ABB RAPID module: Robotpaint.mod

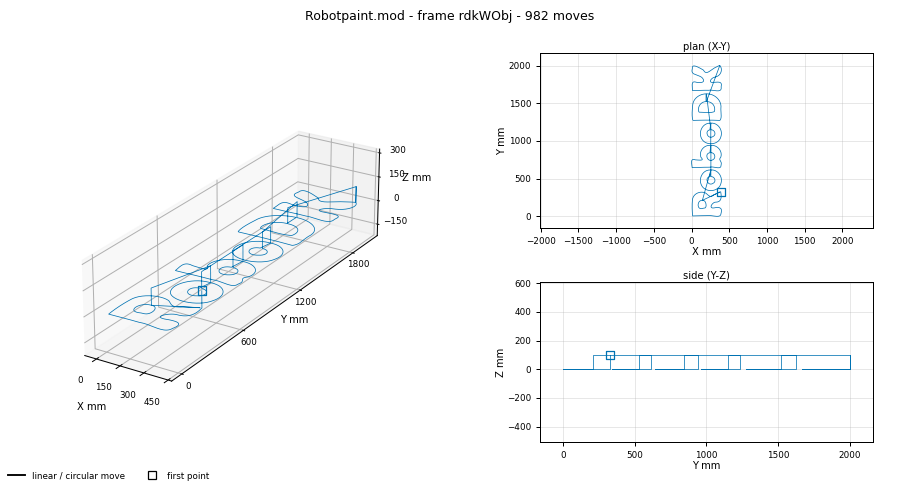
[picture p0: tool path of Robotpaint.mod in frame rdkWObj, 982 of 984 moves have a stored position in this frame; points joined in program order, loops and branches not executed]
MODULE MOD_Robotpaint

PERS wobjdata rdkWObj := [FALSE, TRUE, "", [[0,0,0],[1,0,0,0]],[[0,0,0],[1,0,0,0]]];
PERS tooldata rdkTool := [TRUE,[[0,0,0],[1,0,0,0]],[16,[0,0,15],[1,0,0,0],0,0,0.005]];
VAR speeddata rdkSpeed := [500,500,500,500];
VAR zonedata rdkZone := z0;
VAR extjoint rdkExtax := [9E9,9E9,9E9,9E9,9E9,9E9];

PROC main_RoboDK()
	Robotpaint;
	EXIT;
ENDPROC

PROC Robotpaint()
	!Program generated by RoboDK 2.4.0 for ABB IRB 4600-20/2.50 on 26/06/2016 15:05:34
	!Robot stamp unset
	var robtarget crt;
	crt := CRobT(\Tool:=rdkTool, \WObj:=rdkWObj);
	rdkExtax := crt.extax;
	ConfJ \On;
	ConfL \Off;
	rdkWObj.uframe:=[[0.000,0.000,0.000],[1.00000000,0.00000000,0.00000000,0.00000000]];
	rdkWObj.oframe:=[[1016.501,-940.572,525.712],[1.00000000,0.00000000,0.00000000,0.00000000]];
	rdkTool.tframe:=[[0.000,0.000,283.000],[1.00000000,0.00000000,0.00000000,0.00000000]];
	MoveAbsJ [[0.000000,0.000000,0.000000,0.000000,90.000000,0.000000],rdkExtax], rdkSpeed, rdkZone, rdkTool, \WObj:=rdkWObj;
	MoveL [[386.853,326.209,100.000],[0.00000002,0.00000004,1.00000000,-0.00000004],[-1,-1,-1,0],rdkExtax], rdkSpeed, rdkZone, rdkTool, \WObj:=rdkWObj;
	TPWrite "Drawing path2990";
	SetColorRGB(0.000,0.102,0.655);
	MoveL [[386.853,326.209,0.000],[0.00000002,0.00000004,1.00000000,-0.00000004],[-1,-1,-1,0],rdkExtax], rdkSpeed, rdkZone, rdkTool, \WObj:=rdkWObj;
	MoveL [[388.583,316.262,0.000],[0.00000002,0.00000004,1.00000000,-0.00000004],[-1,-1,-1,0],rdkExtax], rdkSpeed, rdkZone, rdkTool, \WObj:=rdkWObj;
	MoveL [[390.172,306.034,0.000],[0.00000002,0.00000004,1.00000000,-0.00000004],[-1,-1,-1,0],rdkExtax], rdkSpeed, rdkZone, rdkTool, \WObj:=rdkWObj;
	MoveL [[391.529,295.628,0.000],[0.00000002,0.00000004,1.00000000,-0.00000004],[-1,-1,-1,0],rdkExtax], rdkSpeed, rdkZone, rdkTool, \WObj:=rdkWObj;
	MoveL [[392.559,285.148,0.000],[0.00000002,0.00000004,1.00000000,-0.00000004],[-1,-1,-1,0],rdkExtax], rdkSpeed, rdkZone, rdkTool, \WObj:=rdkWObj;
	MoveL [[393.169,274.697,0.000],[0.00000002,0.00000004,1.00000000,-0.00000004],[-1,-1,-1,0],rdkExtax], rdkSpeed, rdkZone, rdkTool, \WObj:=rdkWObj;
	MoveL [[393.265,264.379,0.000],[0.00000002,0.00000004,1.00000000,-0.00000004],[-1,-1,-1,0],rdkExtax], rdkSpeed, rdkZone, rdkTool, \WObj:=rdkWObj;
	MoveL [[392.754,254.297,0.000],[0.00000002,0.00000004,1.00000000,-0.00000004],[-1,-1,-1,0],rdkExtax], rdkSpeed, rdkZone, rdkTool, \WObj:=rdkWObj;
	MoveL [[391.543,244.554,0.000],[0.00000002,0.00000004,1.00000000,-0.00000004],[-1,-1,-1,0],rdkExtax], rdkSpeed, rdkZone, rdkTool, \WObj:=rdkWObj;
	MoveL [[389.538,235.255,0.000],[0.00000002,0.00000004,1.00000000,-0.00000004],[-1,-1,-1,0],rdkExtax], rdkSpeed, rdkZone, rdkTool, \WObj:=rdkWObj;
	MoveL [[386.644,226.502,0.000],[0.00000002,0.00000004,1.00000000,-0.00000004],[-1,-1,-1,0],rdkExtax], rdkSpeed, rdkZone, rdkTool, \WObj:=rdkWObj;
	MoveL [[382.770,218.400,0.000],[0.00000002,0.00000004,1.00000000,-0.00000004],[-1,-1,-1,0],rdkExtax], rdkSpeed, rdkZone, rdkTool, \WObj:=rdkWObj;
	MoveL [[377.821,211.051,0.000],[0.00000002,0.00000004,1.00000000,-0.00000004],[-1,-1,-1,0],rdkExtax], rdkSpeed, rdkZone, rdkTool, \WObj:=rdkWObj;
	MoveL [[371.704,204.559,0.000],[0.00000002,0.00000004,1.00000000,-0.00000004],[-1,-1,-1,0],rdkExtax], rdkSpeed, rdkZone, rdkTool, \WObj:=rdkWObj;
	MoveL [[364.325,199.028,0.000],[0.00000002,0.00000004,1.00000000,-0.00000004],[-1,-1,-1,0],rdkExtax], rdkSpeed, rdkZone, rdkTool, \WObj:=rdkWObj;
	MoveL [[355.592,194.562,0.000],[0.00000002,0.00000004,1.00000000,-0.00000004],[-1,-1,-1,0],rdkExtax], rdkSpeed, rdkZone, rdkTool, \WObj:=rdkWObj;
	MoveL [[345.409,191.263,0.000],[0.00000002,0.00000004,1.00000000,-0.00000004],[-1,-1,-1,0],rdkExtax], rdkSpeed, rdkZone, rdkTool, \WObj:=rdkWObj;
	MoveL [[333.684,189.235,0.000],[0.00000002,0.00000004,1.00000000,-0.00000004],[-1,-1,-1,0],rdkExtax], rdkSpeed, rdkZone, rdkTool, \WObj:=rdkWObj;
	MoveL [[322.010,188.972,0.000],[0.00000002,0.00000004,1.00000000,-0.00000004],[-1,-1,-1,0],rdkExtax], rdkSpeed, rdkZone, rdkTool, \WObj:=rdkWObj;
	MoveL [[311.530,187.503,0.000],[0.00000002,0.00000004,1.00000000,-0.00000004],[-1,-1,-1,0],rdkExtax], rdkSpeed, rdkZone, rdkTool, \WObj:=rdkWObj;
	MoveL [[301.304,183.833,0.000],[0.00000002,0.00000004,1.00000000,-0.00000004],[-1,-1,-1,0],rdkExtax], rdkSpeed, rdkZone, rdkTool, \WObj:=rdkWObj;
	MoveL [[291.597,178.356,0.000],[0.00000002,0.00000004,1.00000000,-0.00000004],[-1,-1,-1,0],rdkExtax], rdkSpeed, rdkZone, rdkTool, \WObj:=rdkWObj;
	MoveL [[282.679,171.466,0.000],[0.00000002,0.00000004,1.00000000,-0.00000004],[-1,-1,-1,0],rdkExtax], rdkSpeed, rdkZone, rdkTool, \WObj:=rdkWObj;
	MoveL [[274.818,163.557,0.000],[0.00000002,0.00000004,1.00000000,-0.00000004],[-1,-1,-1,0],rdkExtax], rdkSpeed, rdkZone, rdkTool, \WObj:=rdkWObj;
	MoveL [[268.281,155.023,0.000],[0.00000002,0.00000004,1.00000000,-0.00000004],[-1,-1,-1,0],rdkExtax], rdkSpeed, rdkZone, rdkTool, \WObj:=rdkWObj;
	MoveL [[263.337,146.257,0.000],[0.00000002,0.00000004,1.00000000,-0.00000004],[-1,-1,-1,0],rdkExtax], rdkSpeed, rdkZone, rdkTool, \WObj:=rdkWObj;
	MoveL [[260.253,137.654,0.000],[0.00000002,0.00000004,1.00000000,-0.00000004],[-1,-1,-1,0],rdkExtax], rdkSpeed, rdkZone, rdkTool, \WObj:=rdkWObj;
	MoveL [[259.298,129.607,0.000],[0.00000002,0.00000004,1.00000000,-0.00000004],[-1,-1,-1,0],rdkExtax], rdkSpeed, rdkZone, rdkTool, \WObj:=rdkWObj;
	MoveL [[260.740,122.511,0.000],[0.00000002,0.00000004,1.00000000,-0.00000004],[-1,-1,-1,0],rdkExtax], rdkSpeed, rdkZone, rdkTool, \WObj:=rdkWObj;
	MoveL [[264.847,116.759,0.000],[0.00000002,0.00000004,1.00000000,-0.00000004],[-1,-1,-1,0],rdkExtax], rdkSpeed, rdkZone, rdkTool, \WObj:=rdkWObj;
	MoveL [[271.887,112.745,0.000],[0.00000002,0.00000004,1.00000000,-0.00000004],[-1,-1,-1,0],rdkExtax], rdkSpeed, rdkZone, rdkTool, \WObj:=rdkWObj;
	MoveL [[282.127,110.864,0.000],[0.00000002,0.00000004,1.00000000,-0.00000004],[-1,-1,-1,0],rdkExtax], rdkSpeed, rdkZone, rdkTool, \WObj:=rdkWObj;
	MoveL [[295.837,111.508,0.000],[0.00000002,0.00000004,1.00000000,-0.00000004],[-1,-1,-1,0],rdkExtax], rdkSpeed, rdkZone, rdkTool, \WObj:=rdkWObj;
	MoveL [[307.788,114.039,0.000],[0.00000002,0.00000004,1.00000000,-0.00000004],[-1,-1,-1,0],rdkExtax], rdkSpeed, rdkZone, rdkTool, \WObj:=rdkWObj;
	MoveL [[319.169,116.073,0.000],[0.00000002,0.00000004,1.00000000,-0.00000004],[-1,-1,-1,0],rdkExtax], rdkSpeed, rdkZone, rdkTool, \WObj:=rdkWObj;
	MoveL [[330.196,117.477,0.000],[0.00000002,0.00000004,1.00000000,-0.00000004],[-1,-1,-1,0],rdkExtax], rdkSpeed, rdkZone, rdkTool, \WObj:=rdkWObj;
	MoveL [[340.758,118.171,0.000],[0.00000002,0.00000004,1.00000000,-0.00000004],[-1,-1,-1,0],rdkExtax], rdkSpeed, rdkZone, rdkTool, \WObj:=rdkWObj;
	MoveL [[350.747,118.075,0.000],[0.00000002,0.00000004,1.00000000,-0.00000004],[-1,-1,-1,0],rdkExtax], rdkSpeed, rdkZone, rdkTool, \WObj:=rdkWObj;
	MoveL [[360.054,117.109,0.000],[0.00000002,0.00000004,1.00000000,-0.00000004],[-1,-1,-1,0],rdkExtax], rdkSpeed, rdkZone, rdkTool, \WObj:=rdkWObj;
	MoveL [[368.570,115.193,0.000],[0.00000002,0.00000004,1.00000000,-0.00000004],[-1,-1,-1,0],rdkExtax], rdkSpeed, rdkZone, rdkTool, \WObj:=rdkWObj;
	MoveL [[376.186,112.248,0.000],[0.00000002,0.00000004,1.00000000,-0.00000004],[-1,-1,-1,0],rdkExtax], rdkSpeed, rdkZone, rdkTool, \WObj:=rdkWObj;
	MoveL [[382.792,108.193,0.000],[0.00000002,0.00000004,1.00000000,-0.00000004],[-1,-1,-1,0],rdkExtax], rdkSpeed, rdkZone, rdkTool, \WObj:=rdkWObj;
	MoveL [[388.280,102.949,0.000],[0.00000002,0.00000004,1.00000000,-0.00000004],[-1,-1,-1,0],rdkExtax], rdkSpeed, rdkZone, rdkTool, \WObj:=rdkWObj;
	MoveL [[392.540,96.436,0.000],[0.00000002,0.00000004,1.00000000,-0.00000004],[-1,-1,-1,0],rdkExtax], rdkSpeed, rdkZone, rdkTool, \WObj:=rdkWObj;
	MoveL [[395.464,88.573,0.000],[0.00000002,0.00000004,1.00000000,-0.00000004],[-1,-1,-1,0],rdkExtax], rdkSpeed, rdkZone, rdkTool, \WObj:=rdkWObj;
	MoveL [[396.942,79.282,0.000],[0.00000002,0.00000004,1.00000000,-0.00000004],[-1,-1,-1,0],rdkExtax], rdkSpeed, rdkZone, rdkTool, \WObj:=rdkWObj;
	MoveL [[396.865,68.481,0.000],[0.00000002,0.00000004,1.00000000,-0.00000004],[-1,-1,-1,0],rdkExtax], rdkSpeed, rdkZone, rdkTool, \WObj:=rdkWObj;
	MoveL [[395.125,56.092,0.000],[0.00000002,0.00000004,1.00000000,-0.00000004],[-1,-1,-1,0],rdkExtax], rdkSpeed, rdkZone, rdkTool, \WObj:=rdkWObj;
	MoveL [[391.611,42.034,0.000],[0.00000002,0.00000004,1.00000000,-0.00000004],[-1,-1,-1,0],rdkExtax], rdkSpeed, rdkZone, rdkTool, \WObj:=rdkWObj;
	MoveL [[390.021,30.870,0.000],[0.00000002,0.00000004,1.00000000,-0.00000004],[-1,-1,-1,0],rdkExtax], rdkSpeed, rdkZone, rdkTool, \WObj:=rdkWObj;
	MoveL [[387.309,21.996,0.000],[0.00000002,0.00000004,1.00000000,-0.00000004],[-1,-1,-1,0],rdkExtax], rdkSpeed, rdkZone, rdkTool, \WObj:=rdkWObj;
	MoveL [[383.123,14.869,0.000],[0.00000002,0.00000004,1.00000000,-0.00000004],[-1,-1,-1,0],rdkExtax], rdkSpeed, rdkZone, rdkTool, \WObj:=rdkWObj;
	MoveL [[377.597,9.334,0.000],[0.00000002,0.00000004,1.00000000,-0.00000004],[-1,-1,-1,0],rdkExtax], rdkSpeed, rdkZone, rdkTool, \WObj:=rdkWObj;
	MoveL [[370.862,5.235,0.000],[0.00000002,0.00000004,1.00000000,-0.00000004],[-1,-1,-1,0],rdkExtax], rdkSpeed, rdkZone, rdkTool, \WObj:=rdkWObj;
	MoveL [[363.049,2.417,0.000],[0.00000002,0.00000004,1.00000000,-0.00000004],[-1,-1,-1,0],rdkExtax], rdkSpeed, rdkZone, rdkTool, \WObj:=rdkWObj;
	MoveL [[354.292,0.724,0.000],[0.00000002,0.00000004,1.00000000,-0.00000004],[-1,-1,-1,0],rdkExtax], rdkSpeed, rdkZone, rdkTool, \WObj:=rdkWObj;
	MoveL [[344.721,0.000,0.000],[0.00000002,0.00000004,1.00000000,-0.00000004],[-1,-1,-1,0],rdkExtax], rdkSpeed, rdkZone, rdkTool, \WObj:=rdkWObj;
	MoveL [[334.469,0.090,0.000],[0.00000002,0.00000004,1.00000000,-0.00000004],[-1,-1,-1,0],rdkExtax], rdkSpeed, rdkZone, rdkTool, \WObj:=rdkWObj;
	MoveL [[323.668,0.839,0.000],[0.00000002,0.00000004,1.00000000,-0.00000004],[-1,-1,-1,0],rdkExtax], rdkSpeed, rdkZone, rdkTool, \WObj:=rdkWObj;
	MoveL [[312.450,2.090,0.000],[0.00000002,0.00000004,1.00000000,-0.00000004],[-1,-1,-1,0],rdkExtax], rdkSpeed, rdkZone, rdkTool, \WObj:=rdkWObj;
	MoveL [[300.946,3.689,0.000],[0.00000002,0.00000004,1.00000000,-0.00000004],[-1,-1,-1,0],rdkExtax], rdkSpeed, rdkZone, rdkTool, \WObj:=rdkWObj;
	MoveL [[289.290,5.479,0.000],[0.00000002,0.00000004,1.00000000,-0.00000004],[-1,-1,-1,0],rdkExtax], rdkSpeed, rdkZone, rdkTool, \WObj:=rdkWObj;
	MoveL [[277.611,7.305,0.000],[0.00000002,0.00000004,1.00000000,-0.00000004],[-1,-1,-1,0],rdkExtax], rdkSpeed, rdkZone, rdkTool, \WObj:=rdkWObj;
	MoveL [[266.044,9.012,0.000],[0.00000002,0.00000004,1.00000000,-0.00000004],[-1,-1,-1,0],rdkExtax], rdkSpeed, rdkZone, rdkTool, \WObj:=rdkWObj;
	MoveL [[254.719,10.444,0.000],[0.00000002,0.00000004,1.00000000,-0.00000004],[-1,-1,-1,0],rdkExtax], rdkSpeed, rdkZone, rdkTool, \WObj:=rdkWObj;
	MoveL [[243.769,11.445,0.000],[0.00000002,0.00000004,1.00000000,-0.00000004],[-1,-1,-1,0],rdkExtax], rdkSpeed, rdkZone, rdkTool, \WObj:=rdkWObj;
	MoveL [[233.325,11.860,0.000],[0.00000002,0.00000004,1.00000000,-0.00000004],[-1,-1,-1,0],rdkExtax], rdkSpeed, rdkZone, rdkTool, \WObj:=rdkWObj;
	MoveL [[223.520,11.534,0.000],[0.00000002,0.00000004,1.00000000,-0.00000004],[-1,-1,-1,0],rdkExtax], rdkSpeed, rdkZone, rdkTool, \WObj:=rdkWObj;
	MoveL [[214.485,10.310,0.000],[0.00000002,0.00000004,1.00000000,-0.00000004],[-1,-1,-1,0],rdkExtax], rdkSpeed, rdkZone, rdkTool, \WObj:=rdkWObj;
	MoveL [[205.606,9.028,0.000],[0.00000002,0.00000004,1.00000000,-0.00000004],[-1,-1,-1,0],rdkExtax], rdkSpeed, rdkZone, rdkTool, \WObj:=rdkWObj;
	MoveL [[195.574,9.230,0.000],[0.00000002,0.00000004,1.00000000,-0.00000004],[-1,-1,-1,0],rdkExtax], rdkSpeed, rdkZone, rdkTool, \WObj:=rdkWObj;
	MoveL [[185.522,9.322,0.000],[0.00000002,0.00000004,1.00000000,-0.00000004],[-1,-1,-1,0],rdkExtax], rdkSpeed, rdkZone, rdkTool, \WObj:=rdkWObj;
	MoveL [[175.452,9.314,0.000],[0.00000002,0.00000004,1.00000000,-0.00000004],[-1,-1,-1,0],rdkExtax], rdkSpeed, rdkZone, rdkTool, \WObj:=rdkWObj;
	MoveL [[165.368,9.219,0.000],[0.00000002,0.00000004,1.00000000,-0.00000004],[-1,-1,-1,0],rdkExtax], rdkSpeed, rdkZone, rdkTool, \WObj:=rdkWObj;
	MoveL [[155.274,9.049,0.000],[0.00000002,0.00000004,1.00000000,-0.00000004],[-1,-1,-1,0],rdkExtax], rdkSpeed, rdkZone, rdkTool, \WObj:=rdkWObj;
	MoveL [[145.172,8.816,0.000],[0.00000002,0.00000004,1.00000000,-0.00000004],[-1,-1,-1,0],rdkExtax], rdkSpeed, rdkZone, rdkTool, \WObj:=rdkWObj;
	MoveL [[135.066,8.532,0.000],[0.00000002,0.00000004,1.00000000,-0.00000004],[-1,-1,-1,0],rdkExtax], rdkSpeed, rdkZone, rdkTool, \WObj:=rdkWObj;
	MoveL [[124.961,8.210,0.000],[0.00000002,0.00000004,1.00000000,-0.00000004],[-1,-1,-1,0],rdkExtax], rdkSpeed, rdkZone, rdkTool, \WObj:=rdkWObj;
	MoveL [[114.858,7.860,0.000],[0.00000002,0.00000004,1.00000000,-0.00000004],[-1,-1,-1,0],rdkExtax], rdkSpeed, rdkZone, rdkTool, \WObj:=rdkWObj;
	MoveL [[104.762,7.496,0.000],[0.00000002,0.00000004,1.00000000,-0.00000004],[-1,-1,-1,0],rdkExtax], rdkSpeed, rdkZone, rdkTool, \WObj:=rdkWObj;
	MoveL [[94.676,7.130,0.000],[0.00000002,0.00000004,1.00000000,-0.00000004],[-1,-1,-1,0],rdkExtax], rdkSpeed, rdkZone, rdkTool, \WObj:=rdkWObj;
	MoveL [[84.604,6.772,0.000],[0.00000002,0.00000004,1.00000000,-0.00000004],[-1,-1,-1,0],rdkExtax], rdkSpeed, rdkZone, rdkTool, \WObj:=rdkWObj;
	MoveL [[74.548,6.437,0.000],[0.00000002,0.00000004,1.00000000,-0.00000004],[-1,-1,-1,0],rdkExtax], rdkSpeed, rdkZone, rdkTool, \WObj:=rdkWObj;
	MoveL [[64.513,6.135,0.000],[0.00000002,0.00000004,1.00000000,-0.00000004],[-1,-1,-1,0],rdkExtax], rdkSpeed, rdkZone, rdkTool, \WObj:=rdkWObj;
	MoveL [[54.502,5.879,0.000],[0.00000002,0.00000004,1.00000000,-0.00000004],[-1,-1,-1,0],rdkExtax], rdkSpeed, rdkZone, rdkTool, \WObj:=rdkWObj;
	MoveL [[44.518,5.681,0.000],[0.00000002,0.00000004,1.00000000,-0.00000004],[-1,-1,-1,0],rdkExtax], rdkSpeed, rdkZone, rdkTool, \WObj:=rdkWObj;
	MoveL [[34.564,5.552,0.000],[0.00000002,0.00000004,1.00000000,-0.00000004],[-1,-1,-1,0],rdkExtax], rdkSpeed, rdkZone, rdkTool, \WObj:=rdkWObj;
	MoveL [[24.645,5.506,0.000],[0.00000002,0.00000004,1.00000000,-0.00000004],[-1,-1,-1,0],rdkExtax], rdkSpeed, rdkZone, rdkTool, \WObj:=rdkWObj;
	MoveL [[14.763,5.553,0.000],[0.00000002,0.00000004,1.00000000,-0.00000004],[-1,-1,-1,0],rdkExtax], rdkSpeed, rdkZone, rdkTool, \WObj:=rdkWObj;
	MoveL [[13.513,15.248,0.000],[0.00000002,0.00000004,1.00000000,-0.00000004],[-1,-1,-1,0],rdkExtax], rdkSpeed, rdkZone, rdkTool, \WObj:=rdkWObj;
	MoveL [[12.534,25.178,0.000],[0.00000002,0.00000004,1.00000000,-0.00000004],[-1,-1,-1,0],rdkExtax], rdkSpeed, rdkZone, rdkTool, \WObj:=rdkWObj;
	MoveL [[11.645,35.139,0.000],[0.00000002,0.00000004,1.00000000,-0.00000004],[-1,-1,-1,0],rdkExtax], rdkSpeed, rdkZone, rdkTool, \WObj:=rdkWObj;
	MoveL [[10.847,45.127,0.000],[0.00000002,0.00000004,1.00000000,-0.00000004],[-1,-1,-1,0],rdkExtax], rdkSpeed, rdkZone, rdkTool, \WObj:=rdkWObj;
	MoveL [[10.140,55.138,0.000],[0.00000002,0.00000004,1.00000000,-0.00000004],[-1,-1,-1,0],rdkExtax], rdkSpeed, rdkZone, rdkTool, \WObj:=rdkWObj;
	MoveL [[9.524,65.170,0.000],[0.00000002,0.00000004,1.00000000,-0.00000004],[-1,-1,-1,0],rdkExtax], rdkSpeed, rdkZone, rdkTool, \WObj:=rdkWObj;
	MoveL [[9.001,75.220,0.000],[0.00000002,0.00000004,1.00000000,-0.00000004],[-1,-1,-1,0],rdkExtax], rdkSpeed, rdkZone, rdkTool, \WObj:=rdkWObj;
	MoveL [[8.570,85.284,0.000],[0.00000002,0.00000004,1.00000000,-0.00000004],[-1,-1,-1,0],rdkExtax], rdkSpeed, rdkZone, rdkTool, \WObj:=rdkWObj;
	MoveL [[8.232,95.359,0.000],[0.00000002,0.00000004,1.00000000,-0.00000004],[-1,-1,-1,0],rdkExtax], rdkSpeed, rdkZone, rdkTool, \WObj:=rdkWObj;
	MoveL [[7.987,105.441,0.000],[0.00000002,0.00000004,1.00000000,-0.00000004],[-1,-1,-1,0],rdkExtax], rdkSpeed, rdkZone, rdkTool, \WObj:=rdkWObj;
	MoveL [[7.837,115.529,0.000],[0.00000002,0.00000004,1.00000000,-0.00000004],[-1,-1,-1,0],rdkExtax], rdkSpeed, rdkZone, rdkTool, \WObj:=rdkWObj;
	MoveL [[7.781,125.619,0.000],[0.00000002,0.00000004,1.00000000,-0.00000004],[-1,-1,-1,0],rdkExtax], rdkSpeed, rdkZone, rdkTool, \WObj:=rdkWObj;
	MoveL [[7.820,135.706,0.000],[0.00000002,0.00000004,1.00000000,-0.00000004],[-1,-1,-1,0],rdkExtax], rdkSpeed, rdkZone, rdkTool, \WObj:=rdkWObj;
	MoveL [[7.954,145.790,0.000],[0.00000002,0.00000004,1.00000000,-0.00000004],[-1,-1,-1,0],rdkExtax], rdkSpeed, rdkZone, rdkTool, \WObj:=rdkWObj;
	MoveL [[8.185,155.865,0.000],[0.00000002,0.00000004,1.00000000,-0.00000004],[-1,-1,-1,0],rdkExtax], rdkSpeed, rdkZone, rdkTool, \WObj:=rdkWObj;
	MoveL [[8.511,165.930,0.000],[0.00000002,0.00000004,1.00000000,-0.00000004],[-1,-1,-1,0],rdkExtax], rdkSpeed, rdkZone, rdkTool, \WObj:=rdkWObj;
	MoveL [[8.935,175.980,0.000],[0.00000002,0.00000004,1.00000000,-0.00000004],[-1,-1,-1,0],rdkExtax], rdkSpeed, rdkZone, rdkTool, \WObj:=rdkWObj;
	MoveL [[9.456,186.013,0.000],[0.00000002,0.00000004,1.00000000,-0.00000004],[-1,-1,-1,0],rdkExtax], rdkSpeed, rdkZone, rdkTool, \WObj:=rdkWObj;
	MoveL [[10.075,196.026,0.000],[0.00000002,0.00000004,1.00000000,-0.00000004],[-1,-1,-1,0],rdkExtax], rdkSpeed, rdkZone, rdkTool, \WObj:=rdkWObj;
	MoveL [[10.792,206.015,0.000],[0.00000002,0.00000004,1.00000000,-0.00000004],[-1,-1,-1,0],rdkExtax], rdkSpeed, rdkZone, rdkTool, \WObj:=rdkWObj;
	MoveL [[11.609,215.978,0.000],[0.00000002,0.00000004,1.00000000,-0.00000004],[-1,-1,-1,0],rdkExtax], rdkSpeed, rdkZone, rdkTool, \WObj:=rdkWObj;
	MoveL [[12.935,226.588,0.000],[0.00000002,0.00000004,1.00000000,-0.00000004],[-1,-1,-1,0],rdkExtax], rdkSpeed, rdkZone, rdkTool, \WObj:=rdkWObj;
	MoveL [[15.233,236.896,0.000],[0.00000002,0.00000004,1.00000000,-0.00000004],[-1,-1,-1,0],rdkExtax], rdkSpeed, rdkZone, rdkTool, \WObj:=rdkWObj;
	MoveL [[18.433,246.681,0.000],[0.00000002,0.00000004,1.00000000,-0.00000004],[-1,-1,-1,0],rdkExtax], rdkSpeed, rdkZone, rdkTool, \WObj:=rdkWObj;
	MoveL [[22.481,255.928,0.000],[0.00000002,0.00000004,1.00000000,-0.00000004],[-1,-1,-1,0],rdkExtax], rdkSpeed, rdkZone, rdkTool, \WObj:=rdkWObj;
	MoveL [[27.320,264.622,0.000],[0.00000002,0.00000004,1.00000000,-0.00000004],[-1,-1,-1,0],rdkExtax], rdkSpeed, rdkZone, rdkTool, \WObj:=rdkWObj;
	MoveL [[32.894,272.749,0.000],[0.00000002,0.00000004,1.00000000,-0.00000004],[-1,-1,-1,0],rdkExtax], rdkSpeed, rdkZone, rdkTool, \WObj:=rdkWObj;
	MoveL [[39.148,280.295,0.000],[0.00000002,0.00000004,1.00000000,-0.00000004],[-1,-1,-1,0],rdkExtax], rdkSpeed, rdkZone, rdkTool, \WObj:=rdkWObj;
	MoveL [[46.026,287.243,0.000],[0.00000002,0.00000004,1.00000000,-0.00000004],[-1,-1,-1,0],rdkExtax], rdkSpeed, rdkZone, rdkTool, \WObj:=rdkWObj;
	MoveL [[53.472,293.581,0.000],[0.00000002,0.00000004,1.00000000,-0.00000004],[-1,-1,-1,0],rdkExtax], rdkSpeed, rdkZone, rdkTool, \WObj:=rdkWObj;
	MoveL [[61.430,299.293,0.000],[0.00000002,0.00000004,1.00000000,-0.00000004],[-1,-1,-1,0],rdkExtax], rdkSpeed, rdkZone, rdkTool, \WObj:=rdkWObj;
	MoveL [[69.845,304.365,0.000],[0.00000002,0.00000004,1.00000000,-0.00000004],[-1,-1,-1,0],rdkExtax], rdkSpeed, rdkZone, rdkTool, \WObj:=rdkWObj;
	MoveL [[78.660,308.781,0.000],[0.00000002,0.00000004,1.00000000,-0.00000004],[-1,-1,-1,0],rdkExtax], rdkSpeed, rdkZone, rdkTool, \WObj:=rdkWObj;
	MoveL [[87.820,312.529,0.000],[0.00000002,0.00000004,1.00000000,-0.00000004],[-1,-1,-1,0],rdkExtax], rdkSpeed, rdkZone, rdkTool, \WObj:=rdkWObj;
	MoveL [[97.270,315.591,0.000],[0.00000002,0.00000004,1.00000000,-0.00000004],[-1,-1,-1,0],rdkExtax], rdkSpeed, rdkZone, rdkTool, \WObj:=rdkWObj;
	MoveL [[106.952,317.955,0.000],[0.00000002,0.00000004,1.00000000,-0.00000004],[-1,-1,-1,0],rdkExtax], rdkSpeed, rdkZone, rdkTool, \WObj:=rdkWObj;
	MoveL [[116.812,319.606,0.000],[0.00000002,0.00000004,1.00000000,-0.00000004],[-1,-1,-1,0],rdkExtax], rdkSpeed, rdkZone, rdkTool, \WObj:=rdkWObj;
	MoveL [[126.793,320.529,0.000],[0.00000002,0.00000004,1.00000000,-0.00000004],[-1,-1,-1,0],rdkExtax], rdkSpeed, rdkZone, rdkTool, \WObj:=rdkWObj;
	MoveL [[136.840,320.708,0.000],[0.00000002,0.00000004,1.00000000,-0.00000004],[-1,-1,-1,0],rdkExtax], rdkSpeed, rdkZone, rdkTool, \WObj:=rdkWObj;
	MoveL [[146.897,320.131,0.000],[0.00000002,0.00000004,1.00000000,-0.00000004],[-1,-1,-1,0],rdkExtax], rdkSpeed, rdkZone, rdkTool, \WObj:=rdkWObj;
	MoveL [[156.909,318.781,0.000],[0.00000002,0.00000004,1.00000000,-0.00000004],[-1,-1,-1,0],rdkExtax], rdkSpeed, rdkZone, rdkTool, \WObj:=rdkWObj;
	MoveL [[166.819,316.645,0.000],[0.00000002,0.00000004,1.00000000,-0.00000004],[-1,-1,-1,0],rdkExtax], rdkSpeed, rdkZone, rdkTool, \WObj:=rdkWObj;
	MoveL [[176.571,313.708,0.000],[0.00000002,0.00000004,1.00000000,-0.00000004],[-1,-1,-1,0],rdkExtax], rdkSpeed, rdkZone, rdkTool, \WObj:=rdkWObj;
	MoveL [[186.110,309.955,0.000],[0.00000002,0.00000004,1.00000000,-0.00000004],[-1,-1,-1,0],rdkExtax], rdkSpeed, rdkZone, rdkTool, \WObj:=rdkWObj;
	MoveL [[194.888,303.784,0.000],[0.00000002,0.00000004,1.00000000,-0.00000004],[-1,-1,-1,0],rdkExtax], rdkSpeed, rdkZone, rdkTool, \WObj:=rdkWObj;
	MoveL [[203.002,296.441,0.000],[0.00000002,0.00000004,1.00000000,-0.00000004],[-1,-1,-1,0],rdkExtax], rdkSpeed, rdkZone, rdkTool, \WObj:=rdkWObj;
	MoveL [[210.818,289.261,0.000],[0.00000002,0.00000004,1.00000000,-0.00000004],[-1,-1,-1,0],rdkExtax], rdkSpeed, rdkZone, rdkTool, \WObj:=rdkWObj;
	MoveL [[218.441,282.511,0.000],[0.00000002,0.00000004,1.00000000,-0.00000004],[-1,-1,-1,0],rdkExtax], rdkSpeed, rdkZone, rdkTool, \WObj:=rdkWObj;
	MoveL [[225.972,276.459,0.000],[0.00000002,0.00000004,1.00000000,-0.00000004],[-1,-1,-1,0],rdkExtax], rdkSpeed, rdkZone, rdkTool, \WObj:=rdkWObj;
	MoveL [[233.515,271.369,0.000],[0.00000002,0.00000004,1.00000000,-0.00000004],[-1,-1,-1,0],rdkExtax], rdkSpeed, rdkZone, rdkTool, \WObj:=rdkWObj;
	MoveL [[241.172,267.510,0.000],[0.00000002,0.00000004,1.00000000,-0.00000004],[-1,-1,-1,0],rdkExtax], rdkSpeed, rdkZone, rdkTool, \WObj:=rdkWObj;
	MoveL [[249.045,265.148,0.000],[0.00000002,0.00000004,1.00000000,-0.00000004],[-1,-1,-1,0],rdkExtax], rdkSpeed, rdkZone, rdkTool, \WObj:=rdkWObj;
	MoveL [[257.237,264.549,0.000],[0.00000002,0.00000004,1.00000000,-0.00000004],[-1,-1,-1,0],rdkExtax], rdkSpeed, rdkZone, rdkTool, \WObj:=rdkWObj;
	MoveL [[265.852,265.981,0.000],[0.00000002,0.00000004,1.00000000,-0.00000004],[-1,-1,-1,0],rdkExtax], rdkSpeed, rdkZone, rdkTool, \WObj:=rdkWObj;
	MoveL [[274.990,269.710,0.000],[0.00000002,0.00000004,1.00000000,-0.00000004],[-1,-1,-1,0],rdkExtax], rdkSpeed, rdkZone, rdkTool, \WObj:=rdkWObj;
	MoveL [[284.756,276.002,0.000],[0.00000002,0.00000004,1.00000000,-0.00000004],[-1,-1,-1,0],rdkExtax], rdkSpeed, rdkZone, rdkTool, \WObj:=rdkWObj;
	MoveL [[295.252,285.125,0.000],[0.00000002,0.00000004,1.00000000,-0.00000004],[-1,-1,-1,0],rdkExtax], rdkSpeed, rdkZone, rdkTool, \WObj:=rdkWObj;
	MoveL [[304.372,289.576,0.000],[0.00000002,0.00000004,1.00000000,-0.00000004],[-1,-1,-1,0],rdkExtax], rdkSpeed, rdkZone, rdkTool, \WObj:=rdkWObj;
	MoveL [[313.416,293.955,0.000],[0.00000002,0.00000004,1.00000000,-0.00000004],[-1,-1,-1,0],rdkExtax], rdkSpeed, rdkZone, rdkTool, \WObj:=rdkWObj;
	MoveL [[322.450,298.383,0.000],[0.00000002,0.00000004,1.00000000,-0.00000004],[-1,-1,-1,0],rdkExtax], rdkSpeed, rdkZone, rdkTool, \WObj:=rdkWObj;
	MoveL [[331.492,302.805,0.000],[0.00000002,0.00000004,1.00000000,-0.00000004],[-1,-1,-1,0],rdkExtax], rdkSpeed, rdkZone, rdkTool, \WObj:=rdkWObj;
	MoveL [[340.562,307.169,0.000],[0.00000002,0.00000004,1.00000000,-0.00000004],[-1,-1,-1,0],rdkExtax], rdkSpeed, rdkZone, rdkTool, \WObj:=rdkWObj;
	MoveL [[349.676,311.420,0.000],[0.00000002,0.00000004,1.00000000,-0.00000004],[-1,-1,-1,0],rdkExtax], rdkSpeed, rdkZone, rdkTool, \WObj:=rdkWObj;
	MoveL [[358.855,315.507,0.000],[0.00000002,0.00000004,1.00000000,-0.00000004],[-1,-1,-1,0],rdkExtax], rdkSpeed, rdkZone, rdkTool, \WObj:=rdkWObj;
	MoveL [[368.115,319.375,0.000],[0.00000002,0.00000004,1.00000000,-0.00000004],[-1,-1,-1,0],rdkExtax], rdkSpeed, rdkZone, rdkTool, \WObj:=rdkWObj;
	MoveL [[377.476,322.971,0.000],[0.00000002,0.00000004,1.00000000,-0.00000004],[-1,-1,-1,0],rdkExtax], rdkSpeed, rdkZone, rdkTool, \WObj:=rdkWObj;
	MoveL [[143.721,212.434,0.000],[0.00000002,0.00000004,1.00000000,-0.00000004],[-1,-1,-1,0],rdkExtax], rdkSpeed, rdkZone, rdkTool, \WObj:=rdkWObj;
	MoveL [[132.355,211.836,0.000],[0.00000002,0.00000004,1.00000000,-0.00000004],[-1,-1,-1,0],rdkExtax], rdkSpeed, rdkZone, rdkTool, \WObj:=rdkWObj;
	MoveL [[122.246,209.110,0.000],[0.00000002,0.00000004,1.00000000,-0.00000004],[-1,-1,-1,0],rdkExtax], rdkSpeed, rdkZone, rdkTool, \WObj:=rdkWObj;
	MoveL [[113.402,204.534,0.000],[0.00000002,0.00000004,1.00000000,-0.00000004],[-1,-1,-1,0],rdkExtax], rdkSpeed, rdkZone, rdkTool, \WObj:=rdkWObj;
	MoveL [[105.831,198.387,0.000],[0.00000002,0.00000004,1.00000000,-0.00000004],[-1,-1,-1,0],rdkExtax], rdkSpeed, rdkZone, rdkTool, \WObj:=rdkWObj;
	MoveL [[99.541,190.946,0.000],[0.00000002,0.00000004,1.00000000,-0.00000004],[-1,-1,-1,0],rdkExtax], rdkSpeed, rdkZone, rdkTool, \WObj:=rdkWObj;
	MoveL [[94.540,182.488,0.000],[0.00000002,0.00000004,1.00000000,-0.00000004],[-1,-1,-1,0],rdkExtax], rdkSpeed, rdkZone, rdkTool, \WObj:=rdkWObj;
	MoveL [[90.836,173.293,0.000],[0.00000002,0.00000004,1.00000000,-0.00000004],[-1,-1,-1,0],rdkExtax], rdkSpeed, rdkZone, rdkTool, \WObj:=rdkWObj;
	MoveL [[88.437,163.637,0.000],[0.00000002,0.00000004,1.00000000,-0.00000004],[-1,-1,-1,0],rdkExtax], rdkSpeed, rdkZone, rdkTool, \WObj:=rdkWObj;
	MoveL [[87.351,153.799,0.000],[0.00000002,0.00000004,1.00000000,-0.00000004],[-1,-1,-1,0],rdkExtax], rdkSpeed, rdkZone, rdkTool, \WObj:=rdkWObj;
	MoveL [[87.585,144.056,0.000],[0.00000002,0.00000004,1.00000000,-0.00000004],[-1,-1,-1,0],rdkExtax], rdkSpeed, rdkZone, rdkTool, \WObj:=rdkWObj;
	MoveL [[89.149,134.686,0.000],[0.00000002,0.00000004,1.00000000,-0.00000004],[-1,-1,-1,0],rdkExtax], rdkSpeed, rdkZone, rdkTool, \WObj:=rdkWObj;
	MoveL [[92.049,125.968,0.000],[0.00000002,0.00000004,1.00000000,-0.00000004],[-1,-1,-1,0],rdkExtax], rdkSpeed, rdkZone, rdkTool, \WObj:=rdkWObj;
	MoveL [[96.294,118.179,0.000],[0.00000002,0.00000004,1.00000000,-0.00000004],[-1,-1,-1,0],rdkExtax], rdkSpeed, rdkZone, rdkTool, \WObj:=rdkWObj;
	MoveL [[101.892,111.596,0.000],[0.00000002,0.00000004,1.00000000,-0.00000004],[-1,-1,-1,0],rdkExtax], rdkSpeed, rdkZone, rdkTool, \WObj:=rdkWObj;
	MoveL [[108.850,106.499,0.000],[0.00000002,0.00000004,1.00000000,-0.00000004],[-1,-1,-1,0],rdkExtax], rdkSpeed, rdkZone, rdkTool, \WObj:=rdkWObj;
	MoveL [[117.178,103.164,0.000],[0.00000002,0.00000004,1.00000000,-0.00000004],[-1,-1,-1,0],rdkExtax], rdkSpeed, rdkZone, rdkTool, \WObj:=rdkWObj;
	MoveL [[126.882,101.870,0.000],[0.00000002,0.00000004,1.00000000,-0.00000004],[-1,-1,-1,0],rdkExtax], rdkSpeed, rdkZone, rdkTool, \WObj:=rdkWObj;
	MoveL [[137.970,102.894,0.000],[0.00000002,0.00000004,1.00000000,-0.00000004],[-1,-1,-1,0],rdkExtax], rdkSpeed, rdkZone, rdkTool, \WObj:=rdkWObj;
	MoveL [[150.451,106.515,0.000],[0.00000002,0.00000004,1.00000000,-0.00000004],[-1,-1,-1,0],rdkExtax], rdkSpeed, rdkZone, rdkTool, \WObj:=rdkWObj;
	MoveL [[162.573,108.117,0.000],[0.00000002,0.00000004,1.00000000,-0.00000004],[-1,-1,-1,0],rdkExtax], rdkSpeed, rdkZone, rdkTool, \WObj:=rdkWObj;
	MoveL [[171.987,108.400,0.000],[0.00000002,0.00000004,1.00000000,-0.00000004],[-1,-1,-1,0],rdkExtax], rdkSpeed, rdkZone, rdkTool, \WObj:=rdkWObj;
	MoveL [[179.607,111.636,0.000],[0.00000002,0.00000004,1.00000000,-0.00000004],[-1,-1,-1,0],rdkExtax], rdkSpeed, rdkZone, rdkTool, \WObj:=rdkWObj;
	MoveL [[185.496,117.362,0.000],[0.00000002,0.00000004,1.00000000,-0.00000004],[-1,-1,-1,0],rdkExtax], rdkSpeed, rdkZone, rdkTool, \WObj:=rdkWObj;
	MoveL [[189.716,125.119,0.000],[0.00000002,0.00000004,1.00000000,-0.00000004],[-1,-1,-1,0],rdkExtax], rdkSpeed, rdkZone, rdkTool, \WObj:=rdkWObj;
	MoveL [[192.330,134.444,0.000],[0.00000002,0.00000004,1.00000000,-0.00000004],[-1,-1,-1,0],rdkExtax], rdkSpeed, rdkZone, rdkTool, \WObj:=rdkWObj;
	MoveL [[193.400,144.876,0.000],[0.00000002,0.00000004,1.00000000,-0.00000004],[-1,-1,-1,0],rdkExtax], rdkSpeed, rdkZone, rdkTool, \WObj:=rdkWObj;
	MoveL [[192.989,155.953,0.000],[0.00000002,0.00000004,1.00000000,-0.00000004],[-1,-1,-1,0],rdkExtax], rdkSpeed, rdkZone, rdkTool, \WObj:=rdkWObj;
	MoveL [[191.158,167.215,0.000],[0.00000002,0.00000004,1.00000000,-0.00000004],[-1,-1,-1,0],rdkExtax], rdkSpeed, rdkZone, rdkTool, \WObj:=rdkWObj;
	MoveL [[187.971,178.198,0.000],[0.00000002,0.00000004,1.00000000,-0.00000004],[-1,-1,-1,0],rdkExtax], rdkSpeed, rdkZone, rdkTool, \WObj:=rdkWObj;
	MoveL [[183.489,188.443,0.000],[0.00000002,0.00000004,1.00000000,-0.00000004],[-1,-1,-1,0],rdkExtax], rdkSpeed, rdkZone, rdkTool, \WObj:=rdkWObj;
	MoveL [[177.776,197.487,0.000],[0.00000002,0.00000004,1.00000000,-0.00000004],[-1,-1,-1,0],rdkExtax], rdkSpeed, rdkZone, rdkTool, \WObj:=rdkWObj;
	MoveL [[170.892,204.869,0.000],[0.00000002,0.00000004,1.00000000,-0.00000004],[-1,-1,-1,0],rdkExtax], rdkSpeed, rdkZone, rdkTool, \WObj:=rdkWObj;
	MoveL [[162.902,210.128,0.000],[0.00000002,0.00000004,1.00000000,-0.00000004],[-1,-1,-1,0],rdkExtax], rdkSpeed, rdkZone, rdkTool, \WObj:=rdkWObj;
	MoveL [[153.867,212.801,0.000],[0.00000002,0.00000004,1.00000000,-0.00000004],[-1,-1,-1,0],rdkExtax], rdkSpeed, rdkZone, rdkTool, \WObj:=rdkWObj;
	MoveL [[143.849,212.428,0.000],[0.00000002,0.00000004,1.00000000,-0.00000004],[-1,-1,-1,0],rdkExtax], rdkSpeed, rdkZone, rdkTool, \WObj:=rdkWObj;
	MoveL [[143.849,212.428,100.000],[0.00000002,0.00000004,1.00000000,-0.00000004],[-1,-1,-1,0],rdkExtax], rdkSpeed, rdkZone, rdkTool, \WObj:=rdkWObj;
	MoveL [[256.276,615.268,100.000],[0.00000002,0.00000004,1.00000000,-0.00000004],[-1,-1,-1,0],rdkExtax], rdkSpeed, rdkZone, rdkTool, \WObj:=rdkWObj;
	TPWrite "Drawing path2992";
	SetColorRGB(0.655,0.486,0.000);
	MoveL [[256.276,615.268,0.000],[0.00000002,0.00000004,1.00000000,-0.00000004],[-1,-1,-1,0],rdkExtax], rdkSpeed, rdkZone, rdkTool, \WObj:=rdkWObj;
	MoveL [[266.939,615.716,0.000],[0.00000002,0.00000004,1.00000000,-0.00000004],[-1,-1,-1,0],rdkExtax], rdkSpeed, rdkZone, rdkTool, \WObj:=rdkWObj;
	MoveL [[277.362,615.241,0.000],[0.00000002,0.00000004,1.00000000,-0.00000004],[-1,-1,-1,0],rdkExtax], rdkSpeed, rdkZone, rdkTool, \WObj:=rdkWObj;
	MoveL [[287.520,613.888,0.000],[0.00000002,0.00000004,1.00000000,-0.00000004],[-1,-1,-1,0],rdkExtax], rdkSpeed, rdkZone, rdkTool, \WObj:=rdkWObj;
	MoveL [[297.388,611.696,0.000],[0.00000002,0.00000004,1.00000000,-0.00000004],[-1,-1,-1,0],rdkExtax], rdkSpeed, rdkZone, rdkTool, \WObj:=rdkWObj;
	MoveL [[306.939,608.709,0.000],[0.00000002,0.00000004,1.00000000,-0.00000004],[-1,-1,-1,0],rdkExtax], rdkSpeed, rdkZone, rdkTool, \WObj:=rdkWObj;
	MoveL [[316.150,604.968,0.000],[0.00000002,0.00000004,1.00000000,-0.00000004],[-1,-1,-1,0],rdkExtax], rdkSpeed, rdkZone, rdkTool, \WObj:=rdkWObj;
	MoveL [[324.993,600.516,0.000],[0.00000002,0.00000004,1.00000000,-0.00000004],[-1,-1,-1,0],rdkExtax], rdkSpeed, rdkZone, rdkTool, \WObj:=rdkWObj;
	MoveL [[333.445,595.395,0.000],[0.00000002,0.00000004,1.00000000,-0.00000004],[-1,-1,-1,0],rdkExtax], rdkSpeed, rdkZone, rdkTool, \WObj:=rdkWObj;
	MoveL [[341.480,589.645,0.000],[0.00000002,0.00000004,1.00000000,-0.00000004],[-1,-1,-1,0],rdkExtax], rdkSpeed, rdkZone, rdkTool, \WObj:=rdkWObj;
	MoveL [[349.072,583.311,0.000],[0.00000002,0.00000004,1.00000000,-0.00000004],[-1,-1,-1,0],rdkExtax], rdkSpeed, rdkZone, rdkTool, \WObj:=rdkWObj;
	MoveL [[356.196,576.433,0.000],[0.00000002,0.00000004,1.00000000,-0.00000004],[-1,-1,-1,0],rdkExtax], rdkSpeed, rdkZone, rdkTool, \WObj:=rdkWObj;
	MoveL [[362.827,569.053,0.000],[0.00000002,0.00000004,1.00000000,-0.00000004],[-1,-1,-1,0],rdkExtax], rdkSpeed, rdkZone, rdkTool, \WObj:=rdkWObj;
	MoveL [[368.940,561.214,0.000],[0.00000002,0.00000004,1.00000000,-0.00000004],[-1,-1,-1,0],rdkExtax], rdkSpeed, rdkZone, rdkTool, \WObj:=rdkWObj;
	MoveL [[374.509,552.958,0.000],[0.00000002,0.00000004,1.00000000,-0.00000004],[-1,-1,-1,0],rdkExtax], rdkSpeed, rdkZone, rdkTool, \WObj:=rdkWObj;
	MoveL [[379.509,544.327,0.000],[0.00000002,0.00000004,1.00000000,-0.00000004],[-1,-1,-1,0],rdkExtax], rdkSpeed, rdkZone, rdkTool, \WObj:=rdkWObj;
	MoveL [[383.914,535.362,0.000],[0.00000002,0.00000004,1.00000000,-0.00000004],[-1,-1,-1,0],rdkExtax], rdkSpeed, rdkZone, rdkTool, \WObj:=rdkWObj;
	MoveL [[387.700,526.106,0.000],[0.00000002,0.00000004,1.00000000,-0.00000004],[-1,-1,-1,0],rdkExtax], rdkSpeed, rdkZone, rdkTool, \WObj:=rdkWObj;
	MoveL [[390.840,516.601,0.000],[0.00000002,0.00000004,1.00000000,-0.00000004],[-1,-1,-1,0],rdkExtax], rdkSpeed, rdkZone, rdkTool, \WObj:=rdkWObj;
	MoveL [[393.311,506.889,0.000],[0.00000002,0.00000004,1.00000000,-0.00000004],[-1,-1,-1,0],rdkExtax], rdkSpeed, rdkZone, rdkTool, \WObj:=rdkWObj;
	MoveL [[395.085,497.012,0.000],[0.00000002,0.00000004,1.00000000,-0.00000004],[-1,-1,-1,0],rdkExtax], rdkSpeed, rdkZone, rdkTool, \WObj:=rdkWObj;
	MoveL [[396.139,487.012,0.000],[0.00000002,0.00000004,1.00000000,-0.00000004],[-1,-1,-1,0],rdkExtax], rdkSpeed, rdkZone, rdkTool, \WObj:=rdkWObj;
	MoveL [[396.446,476.931,0.000],[0.00000002,0.00000004,1.00000000,-0.00000004],[-1,-1,-1,0],rdkExtax], rdkSpeed, rdkZone, rdkTool, \WObj:=rdkWObj;
	MoveL [[395.982,466.810,0.000],[0.00000002,0.00000004,1.00000000,-0.00000004],[-1,-1,-1,0],rdkExtax], rdkSpeed, rdkZone, rdkTool, \WObj:=rdkWObj;
	MoveL [[394.721,456.693,0.000],[0.00000002,0.00000004,1.00000000,-0.00000004],[-1,-1,-1,0],rdkExtax], rdkSpeed, rdkZone, rdkTool, \WObj:=rdkWObj;
	MoveL [[392.638,446.621,0.000],[0.00000002,0.00000004,1.00000000,-0.00000004],[-1,-1,-1,0],rdkExtax], rdkSpeed, rdkZone, rdkTool, \WObj:=rdkWObj;
	MoveL [[389.707,436.636,0.000],[0.00000002,0.00000004,1.00000000,-0.00000004],[-1,-1,-1,0],rdkExtax], rdkSpeed, rdkZone, rdkTool, \WObj:=rdkWObj;
	MoveL [[386.802,426.216,0.000],[0.00000002,0.00000004,1.00000000,-0.00000004],[-1,-1,-1,0],rdkExtax], rdkSpeed, rdkZone, rdkTool, \WObj:=rdkWObj;
	MoveL [[383.087,416.383,0.000],[0.00000002,0.00000004,1.00000000,-0.00000004],[-1,-1,-1,0],rdkExtax], rdkSpeed, rdkZone, rdkTool, \WObj:=rdkWObj;
	MoveL [[378.597,407.153,0.000],[0.00000002,0.00000004,1.00000000,-0.00000004],[-1,-1,-1,0],rdkExtax], rdkSpeed, rdkZone, rdkTool, \WObj:=rdkWObj;
	MoveL [[373.381,398.526,0.000],[0.00000002,0.00000004,1.00000000,-0.00000004],[-1,-1,-1,0],rdkExtax], rdkSpeed, rdkZone, rdkTool, \WObj:=rdkWObj;
	MoveL [[367.488,390.504,0.000],[0.00000002,0.00000004,1.00000000,-0.00000004],[-1,-1,-1,0],rdkExtax], rdkSpeed, rdkZone, rdkTool, \WObj:=rdkWObj;
	MoveL [[360.970,383.088,0.000],[0.00000002,0.00000004,1.00000000,-0.00000004],[-1,-1,-1,0],rdkExtax], rdkSpeed, rdkZone, rdkTool, \WObj:=rdkWObj;
	MoveL [[353.875,376.280,0.000],[0.00000002,0.00000004,1.00000000,-0.00000004],[-1,-1,-1,0],rdkExtax], rdkSpeed, rdkZone, rdkTool, \WObj:=rdkWObj;
	MoveL [[346.254,370.079,0.000],[0.00000002,0.00000004,1.00000000,-0.00000004],[-1,-1,-1,0],rdkExtax], rdkSpeed, rdkZone, rdkTool, \WObj:=rdkWObj;
	MoveL [[338.156,364.489,0.000],[0.00000002,0.00000004,1.00000000,-0.00000004],[-1,-1,-1,0],rdkExtax], rdkSpeed, rdkZone, rdkTool, \WObj:=rdkWObj;
	MoveL [[329.631,359.509,0.000],[0.00000002,0.00000004,1.00000000,-0.00000004],[-1,-1,-1,0],rdkExtax], rdkSpeed, rdkZone, rdkTool, \WObj:=rdkWObj;
	MoveL [[320.730,355.142,0.000],[0.00000002,0.00000004,1.00000000,-0.00000004],[-1,-1,-1,0],rdkExtax], rdkSpeed, rdkZone, rdkTool, \WObj:=rdkWObj;
	MoveL [[311.501,351.388,0.000],[0.00000002,0.00000004,1.00000000,-0.00000004],[-1,-1,-1,0],rdkExtax], rdkSpeed, rdkZone, rdkTool, \WObj:=rdkWObj;
	MoveL [[301.994,348.248,0.000],[0.00000002,0.00000004,1.00000000,-0.00000004],[-1,-1,-1,0],rdkExtax], rdkSpeed, rdkZone, rdkTool, \WObj:=rdkWObj;
	MoveL [[292.261,345.724,0.000],[0.00000002,0.00000004,1.00000000,-0.00000004],[-1,-1,-1,0],rdkExtax], rdkSpeed, rdkZone, rdkTool, \WObj:=rdkWObj;
	MoveL [[282.349,343.817,0.000],[0.00000002,0.00000004,1.00000000,-0.00000004],[-1,-1,-1,0],rdkExtax], rdkSpeed, rdkZone, rdkTool, \WObj:=rdkWObj;
	MoveL [[272.310,342.529,0.000],[0.00000002,0.00000004,1.00000000,-0.00000004],[-1,-1,-1,0],rdkExtax], rdkSpeed, rdkZone, rdkTool, \WObj:=rdkWObj;
	MoveL [[262.193,341.859,0.000],[0.00000002,0.00000004,1.00000000,-0.00000004],[-1,-1,-1,0],rdkExtax], rdkSpeed, rdkZone, rdkTool, \WObj:=rdkWObj;
	MoveL [[252.047,341.811,0.000],[0.00000002,0.00000004,1.00000000,-0.00000004],[-1,-1,-1,0],rdkExtax], rdkSpeed, rdkZone, rdkTool, \WObj:=rdkWObj;
	MoveL [[241.924,342.384,0.000],[0.00000002,0.00000004,1.00000000,-0.00000004],[-1,-1,-1,0],rdkExtax], rdkSpeed, rdkZone, rdkTool, \WObj:=rdkWObj;
	MoveL [[231.871,343.580,0.000],[0.00000002,0.00000004,1.00000000,-0.00000004],[-1,-1,-1,0],rdkExtax], rdkSpeed, rdkZone, rdkTool, \WObj:=rdkWObj;
	MoveL [[221.941,345.400,0.000],[0.00000002,0.00000004,1.00000000,-0.00000004],[-1,-1,-1,0],rdkExtax], rdkSpeed, rdkZone, rdkTool, \WObj:=rdkWObj;
	MoveL [[212.181,347.846,0.000],[0.00000002,0.00000004,1.00000000,-0.00000004],[-1,-1,-1,0],rdkExtax], rdkSpeed, rdkZone, rdkTool, \WObj:=rdkWObj;
	MoveL [[202.642,350.918,0.000],[0.00000002,0.00000004,1.00000000,-0.00000004],[-1,-1,-1,0],rdkExtax], rdkSpeed, rdkZone, rdkTool, \WObj:=rdkWObj;
	MoveL [[193.374,354.618,0.000],[0.00000002,0.00000004,1.00000000,-0.00000004],[-1,-1,-1,0],rdkExtax], rdkSpeed, rdkZone, rdkTool, \WObj:=rdkWObj;
	MoveL [[184.427,358.948,0.000],[0.00000002,0.00000004,1.00000000,-0.00000004],[-1,-1,-1,0],rdkExtax], rdkSpeed, rdkZone, rdkTool, \WObj:=rdkWObj;
	MoveL [[175.851,363.907,0.000],[0.00000002,0.00000004,1.00000000,-0.00000004],[-1,-1,-1,0],rdkExtax], rdkSpeed, rdkZone, rdkTool, \WObj:=rdkWObj;
	MoveL [[167.695,369.498,0.000],[0.00000002,0.00000004,1.00000000,-0.00000004],[-1,-1,-1,0],rdkExtax], rdkSpeed, rdkZone, rdkTool, \WObj:=rdkWObj;
	MoveL [[160.009,375.722,0.000],[0.00000002,0.00000004,1.00000000,-0.00000004],[-1,-1,-1,0],rdkExtax], rdkSpeed, rdkZone, rdkTool, \WObj:=rdkWObj;
	MoveL [[152.843,382.580,0.000],[0.00000002,0.00000004,1.00000000,-0.00000004],[-1,-1,-1,0],rdkExtax], rdkSpeed, rdkZone, rdkTool, \WObj:=rdkWObj;
	MoveL [[146.247,390.073,0.000],[0.00000002,0.00000004,1.00000000,-0.00000004],[-1,-1,-1,0],rdkExtax], rdkSpeed, rdkZone, rdkTool, \WObj:=rdkWObj;
	MoveL [[140.270,398.202,0.000],[0.00000002,0.00000004,1.00000000,-0.00000004],[-1,-1,-1,0],rdkExtax], rdkSpeed, rdkZone, rdkTool, \WObj:=rdkWObj;
	MoveL [[134.964,406.969,0.000],[0.00000002,0.00000004,1.00000000,-0.00000004],[-1,-1,-1,0],rdkExtax], rdkSpeed, rdkZone, rdkTool, \WObj:=rdkWObj;
	MoveL [[130.376,416.374,0.000],[0.00000002,0.00000004,1.00000000,-0.00000004],[-1,-1,-1,0],rdkExtax], rdkSpeed, rdkZone, rdkTool, \WObj:=rdkWObj;
	MoveL [[126.410,426.093,0.000],[0.00000002,0.00000004,1.00000000,-0.00000004],[-1,-1,-1,0],rdkExtax], rdkSpeed, rdkZone, rdkTool, \WObj:=rdkWObj;
	MoveL [[123.053,435.746,0.000],[0.00000002,0.00000004,1.00000000,-0.00000004],[-1,-1,-1,0],rdkExtax], rdkSpeed, rdkZone, rdkTool, \WObj:=rdkWObj;
	MoveL [[120.473,445.579,0.000],[0.00000002,0.00000004,1.00000000,-0.00000004],[-1,-1,-1,0],rdkExtax], rdkSpeed, rdkZone, rdkTool, \WObj:=rdkWObj;
	MoveL [[118.654,455.545,0.000],[0.00000002,0.00000004,1.00000000,-0.00000004],[-1,-1,-1,0],rdkExtax], rdkSpeed, rdkZone, rdkTool, \WObj:=rdkWObj;
	MoveL [[117.577,465.599,0.000],[0.00000002,0.00000004,1.00000000,-0.00000004],[-1,-1,-1,0],rdkExtax], rdkSpeed, rdkZone, rdkTool, \WObj:=rdkWObj;
	MoveL [[117.225,475.694,0.000],[0.00000002,0.00000004,1.00000000,-0.00000004],[-1,-1,-1,0],rdkExtax], rdkSpeed, rdkZone, rdkTool, \WObj:=rdkWObj;
	MoveL [[117.581,485.783,0.000],[0.00000002,0.00000004,1.00000000,-0.00000004],[-1,-1,-1,0],rdkExtax], rdkSpeed, rdkZone, rdkTool, \WObj:=rdkWObj;
	MoveL [[118.627,495.820,0.000],[0.00000002,0.00000004,1.00000000,-0.00000004],[-1,-1,-1,0],rdkExtax], rdkSpeed, rdkZone, rdkTool, \WObj:=rdkWObj;
	MoveL [[120.346,505.758,0.000],[0.00000002,0.00000004,1.00000000,-0.00000004],[-1,-1,-1,0],rdkExtax], rdkSpeed, rdkZone, rdkTool, \WObj:=rdkWObj;
	MoveL [[122.721,515.550,0.000],[0.00000002,0.00000004,1.00000000,-0.00000004],[-1,-1,-1,0],rdkExtax], rdkSpeed, rdkZone, rdkTool, \WObj:=rdkWObj;
	MoveL [[125.734,525.150,0.000],[0.00000002,0.00000004,1.00000000,-0.00000004],[-1,-1,-1,0],rdkExtax], rdkSpeed, rdkZone, rdkTool, \WObj:=rdkWObj;
	MoveL [[129.368,534.512,0.000],[0.00000002,0.00000004,1.00000000,-0.00000004],[-1,-1,-1,0],rdkExtax], rdkSpeed, rdkZone, rdkTool, \WObj:=rdkWObj;
	MoveL [[133.606,543.589,0.000],[0.00000002,0.00000004,1.00000000,-0.00000004],[-1,-1,-1,0],rdkExtax], rdkSpeed, rdkZone, rdkTool, \WObj:=rdkWObj;
	MoveL [[138.430,552.334,0.000],[0.00000002,0.00000004,1.00000000,-0.00000004],[-1,-1,-1,0],rdkExtax], rdkSpeed, rdkZone, rdkTool, \WObj:=rdkWObj;
	MoveL [[143.822,560.700,0.000],[0.00000002,0.00000004,1.00000000,-0.00000004],[-1,-1,-1,0],rdkExtax], rdkSpeed, rdkZone, rdkTool, \WObj:=rdkWObj;
	MoveL [[149.767,568.642,0.000],[0.00000002,0.00000004,1.00000000,-0.00000004],[-1,-1,-1,0],rdkExtax], rdkSpeed, rdkZone, rdkTool, \WObj:=rdkWObj;
	MoveL [[156.245,576.113,0.000],[0.00000002,0.00000004,1.00000000,-0.00000004],[-1,-1,-1,0],rdkExtax], rdkSpeed, rdkZone, rdkTool, \WObj:=rdkWObj;
	MoveL [[163.240,583.065,0.000],[0.00000002,0.00000004,1.00000000,-0.00000004],[-1,-1,-1,0],rdkExtax], rdkSpeed, rdkZone, rdkTool, \WObj:=rdkWObj;
	MoveL [[170.734,589.453,0.000],[0.00000002,0.00000004,1.00000000,-0.00000004],[-1,-1,-1,0],rdkExtax], rdkSpeed, rdkZone, rdkTool, \WObj:=rdkWObj;
	MoveL [[178.710,595.230,0.000],[0.00000002,0.00000004,1.00000000,-0.00000004],[-1,-1,-1,0],rdkExtax], rdkSpeed, rdkZone, rdkTool, \WObj:=rdkWObj;
	MoveL [[187.151,600.350,0.000],[0.00000002,0.00000004,1.00000000,-0.00000004],[-1,-1,-1,0],rdkExtax], rdkSpeed, rdkZone, rdkTool, \WObj:=rdkWObj;
	MoveL [[196.040,604.765,0.000],[0.00000002,0.00000004,1.00000000,-0.00000004],[-1,-1,-1,0],rdkExtax], rdkSpeed, rdkZone, rdkTool, \WObj:=rdkWObj;
	MoveL [[205.358,608.430,0.000],[0.00000002,0.00000004,1.00000000,-0.00000004],[-1,-1,-1,0],rdkExtax], rdkSpeed, rdkZone, rdkTool, \WObj:=rdkWObj;
	MoveL [[215.088,611.297,0.000],[0.00000002,0.00000004,1.00000000,-0.00000004],[-1,-1,-1,0],rdkExtax], rdkSpeed, rdkZone, rdkTool, \WObj:=rdkWObj;
	MoveL [[225.214,613.320,0.000],[0.00000002,0.00000004,1.00000000,-0.00000004],[-1,-1,-1,0],rdkExtax], rdkSpeed, rdkZone, rdkTool, \WObj:=rdkWObj;
	MoveL [[235.717,614.453,0.000],[0.00000002,0.00000004,1.00000000,-0.00000004],[-1,-1,-1,0],rdkExtax], rdkSpeed, rdkZone, rdkTool, \WObj:=rdkWObj;
	MoveL [[246.155,614.867,0.000],[0.00000002,0.00000004,1.00000000,-0.00000004],[-1,-1,-1,0],rdkExtax], rdkSpeed, rdkZone, rdkTool, \WObj:=rdkWObj;
	MoveL [[256.222,615.266,0.000],[0.00000002,0.00000004,1.00000000,-0.00000004],[-1,-1,-1,0],rdkExtax], rdkSpeed, rdkZone, rdkTool, \WObj:=rdkWObj;
	MoveL [[242.819,525.645,0.000],[0.00000002,0.00000004,1.00000000,-0.00000004],[-1,-1,-1,0],rdkExtax], rdkSpeed, rdkZone, rdkTool, \WObj:=rdkWObj;
	MoveL [[231.534,522.823,0.000],[0.00000002,0.00000004,1.00000000,-0.00000004],[-1,-1,-1,0],rdkExtax], rdkSpeed, rdkZone, rdkTool, \WObj:=rdkWObj;
	MoveL [[222.396,518.230,0.000],[0.00000002,0.00000004,1.00000000,-0.00000004],[-1,-1,-1,0],rdkExtax], rdkSpeed, rdkZone, rdkTool, \WObj:=rdkWObj;
	MoveL [[215.306,512.153,0.000],[0.00000002,0.00000004,1.00000000,-0.00000004],[-1,-1,-1,0],rdkExtax], rdkSpeed, rdkZone, rdkTool, \WObj:=rdkWObj;
	MoveL [[210.163,504.879,0.000],[0.00000002,0.00000004,1.00000000,-0.00000004],[-1,-1,-1,0],rdkExtax], rdkSpeed, rdkZone, rdkTool, \WObj:=rdkWObj;
	MoveL [[206.867,496.695,0.000],[0.00000002,0.00000004,1.00000000,-0.00000004],[-1,-1,-1,0],rdkExtax], rdkSpeed, rdkZone, rdkTool, \WObj:=rdkWObj;
	MoveL [[205.316,487.888,0.000],[0.00000002,0.00000004,1.00000000,-0.00000004],[-1,-1,-1,0],rdkExtax], rdkSpeed, rdkZone, rdkTool, \WObj:=rdkWObj;
	MoveL [[205.410,478.746,0.000],[0.00000002,0.00000004,1.00000000,-0.00000004],[-1,-1,-1,0],rdkExtax], rdkSpeed, rdkZone, rdkTool, \WObj:=rdkWObj;
	MoveL [[207.048,469.555,0.000],[0.00000002,0.00000004,1.00000000,-0.00000004],[-1,-1,-1,0],rdkExtax], rdkSpeed, rdkZone, rdkTool, \WObj:=rdkWObj;
	MoveL [[210.130,460.604,0.000],[0.00000002,0.00000004,1.00000000,-0.00000004],[-1,-1,-1,0],rdkExtax], rdkSpeed, rdkZone, rdkTool, \WObj:=rdkWObj;
	MoveL [[214.555,452.178,0.000],[0.00000002,0.00000004,1.00000000,-0.00000004],[-1,-1,-1,0],rdkExtax], rdkSpeed, rdkZone, rdkTool, \WObj:=rdkWObj;
	MoveL [[220.222,444.565,0.000],[0.00000002,0.00000004,1.00000000,-0.00000004],[-1,-1,-1,0],rdkExtax], rdkSpeed, rdkZone, rdkTool, \WObj:=rdkWObj;
	MoveL [[227.031,438.053,0.000],[0.00000002,0.00000004,1.00000000,-0.00000004],[-1,-1,-1,0],rdkExtax], rdkSpeed, rdkZone, rdkTool, \WObj:=rdkWObj;
	MoveL [[234.881,432.928,0.000],[0.00000002,0.00000004,1.00000000,-0.00000004],[-1,-1,-1,0],rdkExtax], rdkSpeed, rdkZone, rdkTool, \WObj:=rdkWObj;
	MoveL [[243.671,429.478,0.000],[0.00000002,0.00000004,1.00000000,-0.00000004],[-1,-1,-1,0],rdkExtax], rdkSpeed, rdkZone, rdkTool, \WObj:=rdkWObj;
	MoveL [[253.301,427.990,0.000],[0.00000002,0.00000004,1.00000000,-0.00000004],[-1,-1,-1,0],rdkExtax], rdkSpeed, rdkZone, rdkTool, \WObj:=rdkWObj;
	MoveL [[263.670,428.750,0.000],[0.00000002,0.00000004,1.00000000,-0.00000004],[-1,-1,-1,0],rdkExtax], rdkSpeed, rdkZone, rdkTool, \WObj:=rdkWObj;
	MoveL [[274.677,432.047,0.000],[0.00000002,0.00000004,1.00000000,-0.00000004],[-1,-1,-1,0],rdkExtax], rdkSpeed, rdkZone, rdkTool, \WObj:=rdkWObj;
	MoveL [[286.183,438.076,0.000],[0.00000002,0.00000004,1.00000000,-0.00000004],[-1,-1,-1,0],rdkExtax], rdkSpeed, rdkZone, rdkTool, \WObj:=rdkWObj;
	MoveL [[295.750,444.415,0.000],[0.00000002,0.00000004,1.00000000,-0.00000004],[-1,-1,-1,0],rdkExtax], rdkSpeed, rdkZone, rdkTool, \WObj:=rdkWObj;
	MoveL [[302.816,452.018,0.000],[0.00000002,0.00000004,1.00000000,-0.00000004],[-1,-1,-1,0],rdkExtax], rdkSpeed, rdkZone, rdkTool, \WObj:=rdkWObj;
	MoveL [[307.525,460.563,0.000],[0.00000002,0.00000004,1.00000000,-0.00000004],[-1,-1,-1,0],rdkExtax], rdkSpeed, rdkZone, rdkTool, \WObj:=rdkWObj;
	MoveL [[310.018,469.725,0.000],[0.00000002,0.00000004,1.00000000,-0.00000004],[-1,-1,-1,0],rdkExtax], rdkSpeed, rdkZone, rdkTool, \WObj:=rdkWObj;
	MoveL [[310.438,479.179,0.000],[0.00000002,0.00000004,1.00000000,-0.00000004],[-1,-1,-1,0],rdkExtax], rdkSpeed, rdkZone, rdkTool, \WObj:=rdkWObj;
	MoveL [[308.928,488.601,0.000],[0.00000002,0.00000004,1.00000000,-0.00000004],[-1,-1,-1,0],rdkExtax], rdkSpeed, rdkZone, rdkTool, \WObj:=rdkWObj;
	MoveL [[305.630,497.667,0.000],[0.00000002,0.00000004,1.00000000,-0.00000004],[-1,-1,-1,0],rdkExtax], rdkSpeed, rdkZone, rdkTool, \WObj:=rdkWObj;
	MoveL [[300.686,506.052,0.000],[0.00000002,0.00000004,1.00000000,-0.00000004],[-1,-1,-1,0],rdkExtax], rdkSpeed, rdkZone, rdkTool, \WObj:=rdkWObj;
	MoveL [[294.240,513.431,0.000],[0.00000002,0.00000004,1.00000000,-0.00000004],[-1,-1,-1,0],rdkExtax], rdkSpeed, rdkZone, rdkTool, \WObj:=rdkWObj;
	MoveL [[286.433,519.481,0.000],[0.00000002,0.00000004,1.00000000,-0.00000004],[-1,-1,-1,0],rdkExtax], rdkSpeed, rdkZone, rdkTool, \WObj:=rdkWObj;
	MoveL [[277.409,523.877,0.000],[0.00000002,0.00000004,1.00000000,-0.00000004],[-1,-1,-1,0],rdkExtax], rdkSpeed, rdkZone, rdkTool, \WObj:=rdkWObj;
	MoveL [[267.309,526.295,0.000],[0.00000002,0.00000004,1.00000000,-0.00000004],[-1,-1,-1,0],rdkExtax], rdkSpeed, rdkZone, rdkTool, \WObj:=rdkWObj;
	MoveL [[256.276,526.410,0.000],[0.00000002,0.00000004,1.00000000,-0.00000004],[-1,-1,-1,0],rdkExtax], rdkSpeed, rdkZone, rdkTool, \WObj:=rdkWObj;
	MoveL [[256.276,526.410,100.000],[0.00000002,0.00000004,1.00000000,-0.00000004],[-1,-1,-1,0],rdkExtax], rdkSpeed, rdkZone, rdkTool, \WObj:=rdkWObj;
	MoveL [[257.088,941.983,100.000],[0.00000002,0.00000004,1.00000000,-0.00000004],[0,-1,0,0],rdkExtax], rdkSpeed, rdkZone, rdkTool, \WObj:=rdkWObj;
	TPWrite "Drawing path2994";
	SetColorRGB(0.000,0.655,0.141);
	MoveL [[257.088,941.983,0.000],[0.00000002,0.00000004,1.00000000,-0.00000004],[0,-1,0,0],rdkExtax], rdkSpeed, rdkZone, rdkTool, \WObj:=rdkWObj;
	MoveL [[267.393,942.440,0.000],[0.00000002,0.00000004,1.00000000,-0.00000004],[0,-1,0,0],rdkExtax], rdkSpeed, rdkZone, rdkTool, \WObj:=rdkWObj;
	MoveL [[277.589,941.984,0.000],[0.00000002,0.00000004,1.00000000,-0.00000004],[0,-1,0,0],rdkExtax], rdkSpeed, rdkZone, rdkTool, \WObj:=rdkWObj;
	MoveL [[287.633,940.655,0.000],[0.00000002,0.00000004,1.00000000,-0.00000004],[0,-1,0,0],rdkExtax], rdkSpeed, rdkZone, rdkTool, \WObj:=rdkWObj;
	MoveL [[297.483,938.494,0.000],[0.00000002,0.00000004,1.00000000,-0.00000004],[-1,-1,-1,0],rdkExtax], rdkSpeed, rdkZone, rdkTool, \WObj:=rdkWObj;
	MoveL [[307.097,935.544,0.000],[0.00000002,0.00000004,1.00000000,-0.00000004],[-1,-1,-1,0],rdkExtax], rdkSpeed, rdkZone, rdkTool, \WObj:=rdkWObj;
	MoveL [[316.430,931.845,0.000],[0.00000002,0.00000004,1.00000000,-0.00000004],[-1,-1,-1,0],rdkExtax], rdkSpeed, rdkZone, rdkTool, \WObj:=rdkWObj;
	MoveL [[325.440,927.438,0.000],[0.00000002,0.00000004,1.00000000,-0.00000004],[-1,-1,-1,0],rdkExtax], rdkSpeed, rdkZone, rdkTool, \WObj:=rdkWObj;
	MoveL [[334.085,922.365,0.000],[0.00000002,0.00000004,1.00000000,-0.00000004],[-1,-1,-1,0],rdkExtax], rdkSpeed, rdkZone, rdkTool, \WObj:=rdkWObj;
	MoveL [[342.321,916.666,0.000],[0.00000002,0.00000004,1.00000000,-0.00000004],[-1,-1,-1,0],rdkExtax], rdkSpeed, rdkZone, rdkTool, \WObj:=rdkWObj;
	MoveL [[350.105,910.383,0.000],[0.00000002,0.00000004,1.00000000,-0.00000004],[-1,-1,-1,0],rdkExtax], rdkSpeed, rdkZone, rdkTool, \WObj:=rdkWObj;
	MoveL [[357.395,903.558,0.000],[0.00000002,0.00000004,1.00000000,-0.00000004],[-1,-1,-1,0],rdkExtax], rdkSpeed, rdkZone, rdkTool, \WObj:=rdkWObj;
	MoveL [[364.148,896.230,0.000],[0.00000002,0.00000004,1.00000000,-0.00000004],[-1,-1,-1,0],rdkExtax], rdkSpeed, rdkZone, rdkTool, \WObj:=rdkWObj;
	MoveL [[370.321,888.442,0.000],[0.00000002,0.00000004,1.00000000,-0.00000004],[-1,-1,-1,0],rdkExtax], rdkSpeed, rdkZone, rdkTool, \WObj:=rdkWObj;
	MoveL [[375.870,880.234,0.000],[0.00000002,0.00000004,1.00000000,-0.00000004],[-1,-1,-1,0],rdkExtax], rdkSpeed, rdkZone, rdkTool, \WObj:=rdkWObj;
	MoveL [[380.754,871.648,0.000],[0.00000002,0.00000004,1.00000000,-0.00000004],[-1,-1,-1,0],rdkExtax], rdkSpeed, rdkZone, rdkTool, \WObj:=rdkWObj;
	MoveL [[384.929,862.725,0.000],[0.00000002,0.00000004,1.00000000,-0.00000004],[-1,-1,-1,0],rdkExtax], rdkSpeed, rdkZone, rdkTool, \WObj:=rdkWObj;
	MoveL [[388.352,853.506,0.000],[0.00000002,0.00000004,1.00000000,-0.00000004],[-1,-1,-1,0],rdkExtax], rdkSpeed, rdkZone, rdkTool, \WObj:=rdkWObj;
	MoveL [[390.981,844.032,0.000],[0.00000002,0.00000004,1.00000000,-0.00000004],[-1,-1,-1,0],rdkExtax], rdkSpeed, rdkZone, rdkTool, \WObj:=rdkWObj;
	MoveL [[392.772,834.345,0.000],[0.00000002,0.00000004,1.00000000,-0.00000004],[-1,-1,-1,0],rdkExtax], rdkSpeed, rdkZone, rdkTool, \WObj:=rdkWObj;
	MoveL [[393.683,824.485,0.000],[0.00000002,0.00000004,1.00000000,-0.00000004],[-1,-1,-1,0],rdkExtax], rdkSpeed, rdkZone, rdkTool, \WObj:=rdkWObj;
	MoveL [[393.671,814.494,0.000],[0.00000002,0.00000004,1.00000000,-0.00000004],[-1,-1,-1,0],rdkExtax], rdkSpeed, rdkZone, rdkTool, \WObj:=rdkWObj;
	MoveL [[392.693,804.414,0.000],[0.00000002,0.00000004,1.00000000,-0.00000004],[-1,-1,-1,0],rdkExtax], rdkSpeed, rdkZone, rdkTool, \WObj:=rdkWObj;
	MoveL [[390.706,794.284,0.000],[0.00000002,0.00000004,1.00000000,-0.00000004],[-1,-1,-1,0],rdkExtax], rdkSpeed, rdkZone, rdkTool, \WObj:=rdkWObj;
	MoveL [[387.666,784.147,0.000],[0.00000002,0.00000004,1.00000000,-0.00000004],[-1,-1,-1,0],rdkExtax], rdkSpeed, rdkZone, rdkTool, \WObj:=rdkWObj;
	MoveL [[379.973,774.185,0.000],[0.00000002,0.00000004,1.00000000,-0.00000004],[-1,-1,-1,0],rdkExtax], rdkSpeed, rdkZone, rdkTool, \WObj:=rdkWObj;
	MoveL [[375.252,765.243,0.000],[0.00000002,0.00000004,1.00000000,-0.00000004],[-1,-1,-1,0],rdkExtax], rdkSpeed, rdkZone, rdkTool, \WObj:=rdkWObj;
	MoveL [[374.033,757.097,0.000],[0.00000002,0.00000004,1.00000000,-0.00000004],[-1,-1,-1,0],rdkExtax], rdkSpeed, rdkZone, rdkTool, \WObj:=rdkWObj;
	MoveL [[375.497,749.443,0.000],[0.00000002,0.00000004,1.00000000,-0.00000004],[-1,-1,-1,0],rdkExtax], rdkSpeed, rdkZone, rdkTool, \WObj:=rdkWObj;
	MoveL [[378.824,741.977,0.000],[0.00000002,0.00000004,1.00000000,-0.00000004],[-1,-1,-1,0],rdkExtax], rdkSpeed, rdkZone, rdkTool, \WObj:=rdkWObj;
	MoveL [[383.196,734.393,0.000],[0.00000002,0.00000004,1.00000000,-0.00000004],[-1,-1,-1,0],rdkExtax], rdkSpeed, rdkZone, rdkTool, \WObj:=rdkWObj;
	MoveL [[387.791,726.388,0.000],[0.00000002,0.00000004,1.00000000,-0.00000004],[-1,-1,-1,0],rdkExtax], rdkSpeed, rdkZone, rdkTool, \WObj:=rdkWObj;
	MoveL [[391.792,717.655,0.000],[0.00000002,0.00000004,1.00000000,-0.00000004],[-1,-1,-1,0],rdkExtax], rdkSpeed, rdkZone, rdkTool, \WObj:=rdkWObj;
	MoveL [[394.378,707.892,0.000],[0.00000002,0.00000004,1.00000000,-0.00000004],[-1,-1,-1,0],rdkExtax], rdkSpeed, rdkZone, rdkTool, \WObj:=rdkWObj;
	MoveL [[394.731,696.792,0.000],[0.00000002,0.00000004,1.00000000,-0.00000004],[-1,-1,-1,0],rdkExtax], rdkSpeed, rdkZone, rdkTool, \WObj:=rdkWObj;
	MoveL [[392.031,684.051,0.000],[0.00000002,0.00000004,1.00000000,-0.00000004],[-1,-1,-1,0],rdkExtax], rdkSpeed, rdkZone, rdkTool, \WObj:=rdkWObj;
	MoveL [[390.593,671.595,0.000],[0.00000002,0.00000004,1.00000000,-0.00000004],[-1,-1,-1,0],rdkExtax], rdkSpeed, rdkZone, rdkTool, \WObj:=rdkWObj;
	MoveL [[389.071,662.037,0.000],[0.00000002,0.00000004,1.00000000,-0.00000004],[-1,-1,-1,0],rdkExtax], rdkSpeed, rdkZone, rdkTool, \WObj:=rdkWObj;
	MoveL [[385.508,654.825,0.000],[0.00000002,0.00000004,1.00000000,-0.00000004],[-1,-1,-1,0],rdkExtax], rdkSpeed, rdkZone, rdkTool, \WObj:=rdkWObj;
	MoveL [[380.129,649.695,0.000],[0.00000002,0.00000004,1.00000000,-0.00000004],[-1,-1,-1,0],rdkExtax], rdkSpeed, rdkZone, rdkTool, \WObj:=rdkWObj;
	MoveL [[373.159,646.383,0.000],[0.00000002,0.00000004,1.00000000,-0.00000004],[-1,-1,-1,0],rdkExtax], rdkSpeed, rdkZone, rdkTool, \WObj:=rdkWObj;
	MoveL [[364.823,644.623,0.000],[0.00000002,0.00000004,1.00000000,-0.00000004],[-1,-1,-1,0],rdkExtax], rdkSpeed, rdkZone, rdkTool, \WObj:=rdkWObj;
	MoveL [[355.346,644.152,0.000],[0.00000002,0.00000004,1.00000000,-0.00000004],[-1,-1,-1,0],rdkExtax], rdkSpeed, rdkZone, rdkTool, \WObj:=rdkWObj;
	MoveL [[344.953,644.706,0.000],[0.00000002,0.00000004,1.00000000,-0.00000004],[-1,-1,-1,0],rdkExtax], rdkSpeed, rdkZone, rdkTool, \WObj:=rdkWObj;
	MoveL [[333.869,646.020,0.000],[0.00000002,0.00000004,1.00000000,-0.00000004],[-1,-1,-1,0],rdkExtax], rdkSpeed, rdkZone, rdkTool, \WObj:=rdkWObj;
	MoveL [[322.320,647.830,0.000],[0.00000002,0.00000004,1.00000000,-0.00000004],[-1,-1,-1,0],rdkExtax], rdkSpeed, rdkZone, rdkTool, \WObj:=rdkWObj;
	MoveL [[310.530,649.871,0.000],[0.00000002,0.00000004,1.00000000,-0.00000004],[-1,-1,-1,0],rdkExtax], rdkSpeed, rdkZone, rdkTool, \WObj:=rdkWObj;
	MoveL [[298.724,651.880,0.000],[0.00000002,0.00000004,1.00000000,-0.00000004],[-1,-1,-1,0],rdkExtax], rdkSpeed, rdkZone, rdkTool, \WObj:=rdkWObj;
	MoveL [[287.127,653.592,0.000],[0.00000002,0.00000004,1.00000000,-0.00000004],[-1,-1,-1,0],rdkExtax], rdkSpeed, rdkZone, rdkTool, \WObj:=rdkWObj;
	MoveL [[275.965,654.742,0.000],[0.00000002,0.00000004,1.00000000,-0.00000004],[-1,-1,-1,0],rdkExtax], rdkSpeed, rdkZone, rdkTool, \WObj:=rdkWObj;
	MoveL [[265.463,655.068,0.000],[0.00000002,0.00000004,1.00000000,-0.00000004],[-1,-1,-1,0],rdkExtax], rdkSpeed, rdkZone, rdkTool, \WObj:=rdkWObj;
	MoveL [[255.845,654.303,0.000],[0.00000002,0.00000004,1.00000000,-0.00000004],[-1,-1,-1,0],rdkExtax], rdkSpeed, rdkZone, rdkTool, \WObj:=rdkWObj;
	MoveL [[247.336,652.184,0.000],[0.00000002,0.00000004,1.00000000,-0.00000004],[-1,-1,-1,0],rdkExtax], rdkSpeed, rdkZone, rdkTool, \WObj:=rdkWObj;
	MoveL [[238.042,651.403,0.000],[0.00000002,0.00000004,1.00000000,-0.00000004],[-1,-1,-1,0],rdkExtax], rdkSpeed, rdkZone, rdkTool, \WObj:=rdkWObj;
	MoveL [[228.004,651.594,0.000],[0.00000002,0.00000004,1.00000000,-0.00000004],[-1,-1,-1,0],rdkExtax], rdkSpeed, rdkZone, rdkTool, \WObj:=rdkWObj;
	MoveL [[217.951,651.695,0.000],[0.00000002,0.00000004,1.00000000,-0.00000004],[-1,-1,-1,0],rdkExtax], rdkSpeed, rdkZone, rdkTool, \WObj:=rdkWObj;
	MoveL [[207.883,651.712,0.000],[0.00000002,0.00000004,1.00000000,-0.00000004],[-1,-1,-1,0],rdkExtax], rdkSpeed, rdkZone, rdkTool, \WObj:=rdkWObj;
	MoveL [[197.804,651.653,0.000],[0.00000002,0.00000004,1.00000000,-0.00000004],[-1,-1,-1,0],rdkExtax], rdkSpeed, rdkZone, rdkTool, \WObj:=rdkWObj;
	MoveL [[187.715,651.523,0.000],[0.00000002,0.00000004,1.00000000,-0.00000004],[-1,-1,-1,0],rdkExtax], rdkSpeed, rdkZone, rdkTool, \WObj:=rdkWObj;
	MoveL [[177.619,651.331,0.000],[0.00000002,0.00000004,1.00000000,-0.00000004],[-1,-1,-1,0],rdkExtax], rdkSpeed, rdkZone, rdkTool, \WObj:=rdkWObj;
	MoveL [[167.519,651.082,0.000],[0.00000002,0.00000004,1.00000000,-0.00000004],[-1,-1,-1,0],rdkExtax], rdkSpeed, rdkZone, rdkTool, \WObj:=rdkWObj;
	MoveL [[157.416,650.784,0.000],[0.00000002,0.00000004,1.00000000,-0.00000004],[-1,-1,-1,0],rdkExtax], rdkSpeed, rdkZone, rdkTool, \WObj:=rdkWObj;
	MoveL [[147.312,650.443,0.000],[0.00000002,0.00000004,1.00000000,-0.00000004],[-1,-1,-1,0],rdkExtax], rdkSpeed, rdkZone, rdkTool, \WObj:=rdkWObj;
	MoveL [[137.211,650.066,0.000],[0.00000002,0.00000004,1.00000000,-0.00000004],[-1,-1,-1,0],rdkExtax], rdkSpeed, rdkZone, rdkTool, \WObj:=rdkWObj;
	MoveL [[127.114,649.660,0.000],[0.00000002,0.00000004,1.00000000,-0.00000004],[-1,-1,-1,0],rdkExtax], rdkSpeed, rdkZone, rdkTool, \WObj:=rdkWObj;
	MoveL [[117.025,649.231,0.000],[0.00000002,0.00000004,1.00000000,-0.00000004],[-1,-1,-1,0],rdkExtax], rdkSpeed, rdkZone, rdkTool, \WObj:=rdkWObj;
	MoveL [[106.944,648.787,0.000],[0.00000002,0.00000004,1.00000000,-0.00000004],[-1,-1,-1,0],rdkExtax], rdkSpeed, rdkZone, rdkTool, \WObj:=rdkWObj;
	MoveL [[96.875,648.334,0.000],[0.00000002,0.00000004,1.00000000,-0.00000004],[-1,-1,-1,0],rdkExtax], rdkSpeed, rdkZone, rdkTool, \WObj:=rdkWObj;
	MoveL [[86.819,647.879,0.000],[0.00000002,0.00000004,1.00000000,-0.00000004],[-1,-1,-1,0],rdkExtax], rdkSpeed, rdkZone, rdkTool, \WObj:=rdkWObj;
	MoveL [[76.780,647.428,0.000],[0.00000002,0.00000004,1.00000000,-0.00000004],[-1,-1,-1,0],rdkExtax], rdkSpeed, rdkZone, rdkTool, \WObj:=rdkWObj;
	MoveL [[66.759,646.989,0.000],[0.00000002,0.00000004,1.00000000,-0.00000004],[-1,-1,-1,0],rdkExtax], rdkSpeed, rdkZone, rdkTool, \WObj:=rdkWObj;
	MoveL [[56.758,646.569,0.000],[0.00000002,0.00000004,1.00000000,-0.00000004],[-1,-1,-1,0],rdkExtax], rdkSpeed, rdkZone, rdkTool, \WObj:=rdkWObj;
	MoveL [[46.781,646.173,0.000],[0.00000002,0.00000004,1.00000000,-0.00000004],[-1,-1,-1,0],rdkExtax], rdkSpeed, rdkZone, rdkTool, \WObj:=rdkWObj;
	MoveL [[36.829,645.809,0.000],[0.00000002,0.00000004,1.00000000,-0.00000004],[-1,-1,-1,0],rdkExtax], rdkSpeed, rdkZone, rdkTool, \WObj:=rdkWObj;
	MoveL [[26.905,645.484,0.000],[0.00000002,0.00000004,1.00000000,-0.00000004],[-1,-1,-1,0],rdkExtax], rdkSpeed, rdkZone, rdkTool, \WObj:=rdkWObj;
	MoveL [[17.010,645.204,0.000],[0.00000002,0.00000004,1.00000000,-0.00000004],[-1,-1,-1,0],rdkExtax], rdkSpeed, rdkZone, rdkTool, \WObj:=rdkWObj;
	MoveL [[8.199,645.997,0.000],[0.00000002,0.00000004,1.00000000,-0.00000004],[-1,-1,-1,0],rdkExtax], rdkSpeed, rdkZone, rdkTool, \WObj:=rdkWObj;
	MoveL [[7.302,655.404,0.000],[0.00000002,0.00000004,1.00000000,-0.00000004],[-1,-1,-1,0],rdkExtax], rdkSpeed, rdkZone, rdkTool, \WObj:=rdkWObj;
	MoveL [[5.921,665.638,0.000],[0.00000002,0.00000004,1.00000000,-0.00000004],[-1,-1,-1,0],rdkExtax], rdkSpeed, rdkZone, rdkTool, \WObj:=rdkWObj;
	MoveL [[4.291,676.427,0.000],[0.00000002,0.00000004,1.00000000,-0.00000004],[-1,-1,-1,0],rdkExtax], rdkSpeed, rdkZone, rdkTool, \WObj:=rdkWObj;
	MoveL [[2.649,687.494,0.000],[0.00000002,0.00000004,1.00000000,-0.00000004],[-1,-1,-1,0],rdkExtax], rdkSpeed, rdkZone, rdkTool, \WObj:=rdkWObj;
	MoveL [[1.229,698.568,0.000],[0.00000002,0.00000004,1.00000000,-0.00000004],[-1,-1,-1,0],rdkExtax], rdkSpeed, rdkZone, rdkTool, \WObj:=rdkWObj;
	MoveL [[0.268,709.374,0.000],[0.00000002,0.00000004,1.00000000,-0.00000004],[-1,-1,-1,0],rdkExtax], rdkSpeed, rdkZone, rdkTool, \WObj:=rdkWObj;
	MoveL [[0.000,719.638,0.000],[0.00000002,0.00000004,1.00000000,-0.00000004],[-1,-1,-1,0],rdkExtax], rdkSpeed, rdkZone, rdkTool, \WObj:=rdkWObj;
	MoveL [[0.661,729.086,0.000],[0.00000002,0.00000004,1.00000000,-0.00000004],[-1,-1,-1,0],rdkExtax], rdkSpeed, rdkZone, rdkTool, \WObj:=rdkWObj;
	MoveL [[2.487,737.445,0.000],[0.00000002,0.00000004,1.00000000,-0.00000004],[-1,-1,-1,0],rdkExtax], rdkSpeed, rdkZone, rdkTool, \WObj:=rdkWObj;
	MoveL [[5.713,744.440,0.000],[0.00000002,0.00000004,1.00000000,-0.00000004],[-1,-1,-1,0],rdkExtax], rdkSpeed, rdkZone, rdkTool, \WObj:=rdkWObj;
	MoveL [[10.575,749.798,0.000],[0.00000002,0.00000004,1.00000000,-0.00000004],[-1,-1,-1,0],rdkExtax], rdkSpeed, rdkZone, rdkTool, \WObj:=rdkWObj;
	MoveL [[17.308,753.245,0.000],[0.00000002,0.00000004,1.00000000,-0.00000004],[-1,-1,-1,0],rdkExtax], rdkSpeed, rdkZone, rdkTool, \WObj:=rdkWObj;
	MoveL [[26.148,754.506,0.000],[0.00000002,0.00000004,1.00000000,-0.00000004],[-1,-1,-1,0],rdkExtax], rdkSpeed, rdkZone, rdkTool, \WObj:=rdkWObj;
	MoveL [[37.329,753.308,0.000],[0.00000002,0.00000004,1.00000000,-0.00000004],[-1,-1,-1,0],rdkExtax], rdkSpeed, rdkZone, rdkTool, \WObj:=rdkWObj;
	MoveL [[51.089,749.377,0.000],[0.00000002,0.00000004,1.00000000,-0.00000004],[-1,-1,-1,0],rdkExtax], rdkSpeed, rdkZone, rdkTool, \WObj:=rdkWObj;
	MoveL [[61.502,748.124,0.000],[0.00000002,0.00000004,1.00000000,-0.00000004],[-1,-1,-1,0],rdkExtax], rdkSpeed, rdkZone, rdkTool, \WObj:=rdkWObj;
	MoveL [[71.964,747.623,0.000],[0.00000002,0.00000004,1.00000000,-0.00000004],[-1,-1,-1,0],rdkExtax], rdkSpeed, rdkZone, rdkTool, \WObj:=rdkWObj;
	MoveL [[83.551,746.776,0.000],[0.00000002,0.00000004,1.00000000,-0.00000004],[-1,-1,-1,0],rdkExtax], rdkSpeed, rdkZone, rdkTool, \WObj:=rdkWObj;
	MoveL [[95.623,745.891,0.000],[0.00000002,0.00000004,1.00000000,-0.00000004],[-1,-1,-1,0],rdkExtax], rdkSpeed, rdkZone, rdkTool, \WObj:=rdkWObj;
	MoveL [[107.540,745.273,0.000],[0.00000002,0.00000004,1.00000000,-0.00000004],[-1,-1,-1,0],rdkExtax], rdkSpeed, rdkZone, rdkTool, \WObj:=rdkWObj;
	MoveL [[118.662,745.232,0.000],[0.00000002,0.00000004,1.00000000,-0.00000004],[-1,-1,-1,0],rdkExtax], rdkSpeed, rdkZone, rdkTool, \WObj:=rdkWObj;
	MoveL [[128.349,746.072,0.000],[0.00000002,0.00000004,1.00000000,-0.00000004],[-1,-1,-1,0],rdkExtax], rdkSpeed, rdkZone, rdkTool, \WObj:=rdkWObj;
	MoveL [[135.963,748.101,0.000],[0.00000002,0.00000004,1.00000000,-0.00000004],[-1,-1,-1,0],rdkExtax], rdkSpeed, rdkZone, rdkTool, \WObj:=rdkWObj;
	MoveL [[140.862,751.627,0.000],[0.00000002,0.00000004,1.00000000,-0.00000004],[-1,-1,-1,0],rdkExtax], rdkSpeed, rdkZone, rdkTool, \WObj:=rdkWObj;
	MoveL [[142.408,756.955,0.000],[0.00000002,0.00000004,1.00000000,-0.00000004],[-1,-1,-1,0],rdkExtax], rdkSpeed, rdkZone, rdkTool, \WObj:=rdkWObj;
	MoveL [[139.960,764.394,0.000],[0.00000002,0.00000004,1.00000000,-0.00000004],[-1,-1,-1,0],rdkExtax], rdkSpeed, rdkZone, rdkTool, \WObj:=rdkWObj;
	MoveL [[132.879,774.249,0.000],[0.00000002,0.00000004,1.00000000,-0.00000004],[-1,-1,-1,0],rdkExtax], rdkSpeed, rdkZone, rdkTool, \WObj:=rdkWObj;
	MoveL [[123.736,785.727,0.000],[0.00000002,0.00000004,1.00000000,-0.00000004],[-1,-1,-1,0],rdkExtax], rdkSpeed, rdkZone, rdkTool, \WObj:=rdkWObj;
	MoveL [[120.665,795.748,0.000],[0.00000002,0.00000004,1.00000000,-0.00000004],[-1,-1,-1,0],rdkExtax], rdkSpeed, rdkZone, rdkTool, \WObj:=rdkWObj;
	MoveL [[118.638,805.803,0.000],[0.00000002,0.00000004,1.00000000,-0.00000004],[-1,-1,-1,0],rdkExtax], rdkSpeed, rdkZone, rdkTool, \WObj:=rdkWObj;
	MoveL [[117.614,815.845,0.000],[0.00000002,0.00000004,1.00000000,-0.00000004],[-1,-1,-1,0],rdkExtax], rdkSpeed, rdkZone, rdkTool, \WObj:=rdkWObj;
	MoveL [[117.552,825.826,0.000],[0.00000002,0.00000004,1.00000000,-0.00000004],[-1,-1,-1,0],rdkExtax], rdkSpeed, rdkZone, rdkTool, \WObj:=rdkWObj;
	MoveL [[118.411,835.700,0.000],[0.00000002,0.00000004,1.00000000,-0.00000004],[-1,-1,-1,0],rdkExtax], rdkSpeed, rdkZone, rdkTool, \WObj:=rdkWObj;
	MoveL [[120.149,845.419,0.000],[0.00000002,0.00000004,1.00000000,-0.00000004],[-1,-1,-1,0],rdkExtax], rdkSpeed, rdkZone, rdkTool, \WObj:=rdkWObj;
	MoveL [[122.727,854.937,0.000],[0.00000002,0.00000004,1.00000000,-0.00000004],[-1,-1,-1,0],rdkExtax], rdkSpeed, rdkZone, rdkTool, \WObj:=rdkWObj;
	MoveL [[126.102,864.206,0.000],[0.00000002,0.00000004,1.00000000,-0.00000004],[-1,-1,-1,0],rdkExtax], rdkSpeed, rdkZone, rdkTool, \WObj:=rdkWObj;
	MoveL [[130.234,873.180,0.000],[0.00000002,0.00000004,1.00000000,-0.00000004],[-1,-1,-1,0],rdkExtax], rdkSpeed, rdkZone, rdkTool, \WObj:=rdkWObj;
	MoveL [[135.082,881.811,0.000],[0.00000002,0.00000004,1.00000000,-0.00000004],[-1,-1,-1,0],rdkExtax], rdkSpeed, rdkZone, rdkTool, \WObj:=rdkWObj;
	MoveL [[140.605,890.051,0.000],[0.00000002,0.00000004,1.00000000,-0.00000004],[-1,-1,-1,0],rdkExtax], rdkSpeed, rdkZone, rdkTool, \WObj:=rdkWObj;
	MoveL [[146.761,897.855,0.000],[0.00000002,0.00000004,1.00000000,-0.00000004],[-1,-1,-1,0],rdkExtax], rdkSpeed, rdkZone, rdkTool, \WObj:=rdkWObj;
	MoveL [[153.511,905.175,0.000],[0.00000002,0.00000004,1.00000000,-0.00000004],[-1,-1,-1,0],rdkExtax], rdkSpeed, rdkZone, rdkTool, \WObj:=rdkWObj;
	MoveL [[160.812,911.964,0.000],[0.00000002,0.00000004,1.00000000,-0.00000004],[-1,-1,-1,0],rdkExtax], rdkSpeed, rdkZone, rdkTool, \WObj:=rdkWObj;
	MoveL [[168.623,918.174,0.000],[0.00000002,0.00000004,1.00000000,-0.00000004],[-1,-1,-1,0],rdkExtax], rdkSpeed, rdkZone, rdkTool, \WObj:=rdkWObj;
	MoveL [[176.905,923.759,0.000],[0.00000002,0.00000004,1.00000000,-0.00000004],[-1,-1,-1,0],rdkExtax], rdkSpeed, rdkZone, rdkTool, \WObj:=rdkWObj;
	MoveL [[185.615,928.671,0.000],[0.00000002,0.00000004,1.00000000,-0.00000004],[-1,-1,-1,0],rdkExtax], rdkSpeed, rdkZone, rdkTool, \WObj:=rdkWObj;
	MoveL [[194.712,932.864,0.000],[0.00000002,0.00000004,1.00000000,-0.00000004],[-1,-1,-1,0],rdkExtax], rdkSpeed, rdkZone, rdkTool, \WObj:=rdkWObj;
	MoveL [[204.157,936.291,0.000],[0.00000002,0.00000004,1.00000000,-0.00000004],[-1,-1,-1,0],rdkExtax], rdkSpeed, rdkZone, rdkTool, \WObj:=rdkWObj;
	MoveL [[213.906,938.904,0.000],[0.00000002,0.00000004,1.00000000,-0.00000004],[-1,-1,-1,0],rdkExtax], rdkSpeed, rdkZone, rdkTool, \WObj:=rdkWObj;
	MoveL [[223.921,940.656,0.000],[0.00000002,0.00000004,1.00000000,-0.00000004],[0,-1,0,0],rdkExtax], rdkSpeed, rdkZone, rdkTool, \WObj:=rdkWObj;
	MoveL [[234.159,941.500,0.000],[0.00000002,0.00000004,1.00000000,-0.00000004],[0,-1,0,0],rdkExtax], rdkSpeed, rdkZone, rdkTool, \WObj:=rdkWObj;
	MoveL [[244.480,941.573,0.000],[0.00000002,0.00000004,1.00000000,-0.00000004],[0,-1,0,0],rdkExtax], rdkSpeed, rdkZone, rdkTool, \WObj:=rdkWObj;
	MoveL [[254.520,941.899,0.000],[0.00000002,0.00000004,1.00000000,-0.00000004],[0,-1,0,0],rdkExtax], rdkSpeed, rdkZone, rdkTool, \WObj:=rdkWObj;
	MoveL [[244.060,843.429,0.000],[0.00000002,0.00000004,1.00000000,-0.00000004],[-1,-1,-1,0],rdkExtax], rdkSpeed, rdkZone, rdkTool, \WObj:=rdkWObj;
	MoveL [[232.435,840.996,0.000],[0.00000002,0.00000004,1.00000000,-0.00000004],[-1,-1,-1,0],rdkExtax], rdkSpeed, rdkZone, rdkTool, \WObj:=rdkWObj;
	MoveL [[222.882,836.768,0.000],[0.00000002,0.00000004,1.00000000,-0.00000004],[-1,-1,-1,0],rdkExtax], rdkSpeed, rdkZone, rdkTool, \WObj:=rdkWObj;
	MoveL [[215.309,831.020,0.000],[0.00000002,0.00000004,1.00000000,-0.00000004],[-1,-1,-1,0],rdkExtax], rdkSpeed, rdkZone, rdkTool, \WObj:=rdkWObj;
	MoveL [[209.625,824.023,0.000],[0.00000002,0.00000004,1.00000000,-0.00000004],[-1,-1,-1,0],rdkExtax], rdkSpeed, rdkZone, rdkTool, \WObj:=rdkWObj;
	MoveL [[205.739,816.051,0.000],[0.00000002,0.00000004,1.00000000,-0.00000004],[-1,-1,-1,0],rdkExtax], rdkSpeed, rdkZone, rdkTool, \WObj:=rdkWObj;
	MoveL [[203.559,807.376,0.000],[0.00000002,0.00000004,1.00000000,-0.00000004],[-1,-1,-1,0],rdkExtax], rdkSpeed, rdkZone, rdkTool, \WObj:=rdkWObj;
	MoveL [[202.995,798.271,0.000],[0.00000002,0.00000004,1.00000000,-0.00000004],[-1,-1,-1,0],rdkExtax], rdkSpeed, rdkZone, rdkTool, \WObj:=rdkWObj;
	MoveL [[203.955,789.009,0.000],[0.00000002,0.00000004,1.00000000,-0.00000004],[-1,-1,-1,0],rdkExtax], rdkSpeed, rdkZone, rdkTool, \WObj:=rdkWObj;
	MoveL [[206.348,779.863,0.000],[0.00000002,0.00000004,1.00000000,-0.00000004],[-1,-1,-1,0],rdkExtax], rdkSpeed, rdkZone, rdkTool, \WObj:=rdkWObj;
	MoveL [[210.082,771.104,0.000],[0.00000002,0.00000004,1.00000000,-0.00000004],[-1,-1,-1,0],rdkExtax], rdkSpeed, rdkZone, rdkTool, \WObj:=rdkWObj;
	MoveL [[215.067,763.007,0.000],[0.00000002,0.00000004,1.00000000,-0.00000004],[-1,-1,-1,0],rdkExtax], rdkSpeed, rdkZone, rdkTool, \WObj:=rdkWObj;
	MoveL [[221.211,755.843,0.000],[0.00000002,0.00000004,1.00000000,-0.00000004],[-1,-1,-1,0],rdkExtax], rdkSpeed, rdkZone, rdkTool, \WObj:=rdkWObj;
	MoveL [[228.423,749.886,0.000],[0.00000002,0.00000004,1.00000000,-0.00000004],[-1,-1,-1,0],rdkExtax], rdkSpeed, rdkZone, rdkTool, \WObj:=rdkWObj;
	MoveL [[236.612,745.408,0.000],[0.00000002,0.00000004,1.00000000,-0.00000004],[-1,-1,-1,0],rdkExtax], rdkSpeed, rdkZone, rdkTool, \WObj:=rdkWObj;
	MoveL [[245.686,742.683,0.000],[0.00000002,0.00000004,1.00000000,-0.00000004],[-1,-1,-1,0],rdkExtax], rdkSpeed, rdkZone, rdkTool, \WObj:=rdkWObj;
	MoveL [[255.554,741.982,0.000],[0.00000002,0.00000004,1.00000000,-0.00000004],[-1,-1,-1,0],rdkExtax], rdkSpeed, rdkZone, rdkTool, \WObj:=rdkWObj;
	MoveL [[266.125,743.579,0.000],[0.00000002,0.00000004,1.00000000,-0.00000004],[-1,-1,-1,0],rdkExtax], rdkSpeed, rdkZone, rdkTool, \WObj:=rdkWObj;
	MoveL [[277.308,747.746,0.000],[0.00000002,0.00000004,1.00000000,-0.00000004],[-1,-1,-1,0],rdkExtax], rdkSpeed, rdkZone, rdkTool, \WObj:=rdkWObj;
	MoveL [[288.337,754.142,0.000],[0.00000002,0.00000004,1.00000000,-0.00000004],[-1,-1,-1,0],rdkExtax], rdkSpeed, rdkZone, rdkTool, \WObj:=rdkWObj;
	MoveL [[296.578,761.144,0.000],[0.00000002,0.00000004,1.00000000,-0.00000004],[-1,-1,-1,0],rdkExtax], rdkSpeed, rdkZone, rdkTool, \WObj:=rdkWObj;
	MoveL [[302.614,769.263,0.000],[0.00000002,0.00000004,1.00000000,-0.00000004],[-1,-1,-1,0],rdkExtax], rdkSpeed, rdkZone, rdkTool, \WObj:=rdkWObj;
	MoveL [[306.553,778.190,0.000],[0.00000002,0.00000004,1.00000000,-0.00000004],[-1,-1,-1,0],rdkExtax], rdkSpeed, rdkZone, rdkTool, \WObj:=rdkWObj;
	MoveL [[308.502,787.616,0.000],[0.00000002,0.00000004,1.00000000,-0.00000004],[-1,-1,-1,0],rdkExtax], rdkSpeed, rdkZone, rdkTool, \WObj:=rdkWObj;
	MoveL [[308.567,797.232,0.000],[0.00000002,0.00000004,1.00000000,-0.00000004],[-1,-1,-1,0],rdkExtax], rdkSpeed, rdkZone, rdkTool, \WObj:=rdkWObj;
	MoveL [[306.856,806.728,0.000],[0.00000002,0.00000004,1.00000000,-0.00000004],[-1,-1,-1,0],rdkExtax], rdkSpeed, rdkZone, rdkTool, \WObj:=rdkWObj;
	MoveL [[303.475,815.797,0.000],[0.00000002,0.00000004,1.00000000,-0.00000004],[-1,-1,-1,0],rdkExtax], rdkSpeed, rdkZone, rdkTool, \WObj:=rdkWObj;
	MoveL [[298.532,824.129,0.000],[0.00000002,0.00000004,1.00000000,-0.00000004],[-1,-1,-1,0],rdkExtax], rdkSpeed, rdkZone, rdkTool, \WObj:=rdkWObj;
	MoveL [[292.132,831.415,0.000],[0.00000002,0.00000004,1.00000000,-0.00000004],[-1,-1,-1,0],rdkExtax], rdkSpeed, rdkZone, rdkTool, \WObj:=rdkWObj;
	MoveL [[284.383,837.345,0.000],[0.00000002,0.00000004,1.00000000,-0.00000004],[-1,-1,-1,0],rdkExtax], rdkSpeed, rdkZone, rdkTool, \WObj:=rdkWObj;
	MoveL [[275.391,841.611,0.000],[0.00000002,0.00000004,1.00000000,-0.00000004],[-1,-1,-1,0],rdkExtax], rdkSpeed, rdkZone, rdkTool, \WObj:=rdkWObj;
	MoveL [[265.264,843.904,0.000],[0.00000002,0.00000004,1.00000000,-0.00000004],[-1,-1,-1,0],rdkExtax], rdkSpeed, rdkZone, rdkTool, \WObj:=rdkWObj;
	MoveL [[254.108,843.914,0.000],[0.00000002,0.00000004,1.00000000,-0.00000004],[-1,-1,-1,0],rdkExtax], rdkSpeed, rdkZone, rdkTool, \WObj:=rdkWObj;
	MoveL [[254.108,843.914,100.000],[0.00000002,0.00000004,1.00000000,-0.00000004],[-1,-1,-1,0],rdkExtax], rdkSpeed, rdkZone, rdkTool, \WObj:=rdkWObj;
	MoveL [[256.276,1236.189,100.000],[0.00000002,0.00000004,1.00000000,-0.00000004],[0,-1,0,0],rdkExtax], rdkSpeed, rdkZone, rdkTool, \WObj:=rdkWObj;
	TPWrite "Drawing path2996";
	SetColorRGB(0.000,0.000,0.000);
	MoveL [[256.276,1236.189,0.000],[0.00000002,0.00000004,1.00000000,-0.00000004],[0,-1,0,0],rdkExtax], rdkSpeed, rdkZone, rdkTool, \WObj:=rdkWObj;
	MoveL [[266.939,1236.636,0.000],[0.00000002,0.00000004,1.00000000,-0.00000004],[0,-1,0,0],rdkExtax], rdkSpeed, rdkZone, rdkTool, \WObj:=rdkWObj;
	MoveL [[277.362,1236.162,0.000],[0.00000002,0.00000004,1.00000000,-0.00000004],[0,-1,0,0],rdkExtax], rdkSpeed, rdkZone, rdkTool, \WObj:=rdkWObj;
	MoveL [[287.520,1234.809,0.000],[0.00000002,0.00000004,1.00000000,-0.00000004],[0,-1,0,0],rdkExtax], rdkSpeed, rdkZone, rdkTool, \WObj:=rdkWObj;
	MoveL [[297.388,1232.617,0.000],[0.00000002,0.00000004,1.00000000,-0.00000004],[0,-1,0,0],rdkExtax], rdkSpeed, rdkZone, rdkTool, \WObj:=rdkWObj;
	MoveL [[306.939,1229.630,0.000],[0.00000002,0.00000004,1.00000000,-0.00000004],[0,-1,0,0],rdkExtax], rdkSpeed, rdkZone, rdkTool, \WObj:=rdkWObj;
	MoveL [[316.150,1225.889,0.000],[0.00000002,0.00000004,1.00000000,-0.00000004],[0,-1,0,0],rdkExtax], rdkSpeed, rdkZone, rdkTool, \WObj:=rdkWObj;
	MoveL [[324.993,1221.437,0.000],[0.00000002,0.00000004,1.00000000,-0.00000004],[0,-1,0,0],rdkExtax], rdkSpeed, rdkZone, rdkTool, \WObj:=rdkWObj;
	MoveL [[333.445,1216.315,0.000],[0.00000002,0.00000004,1.00000000,-0.00000004],[0,-1,0,0],rdkExtax], rdkSpeed, rdkZone, rdkTool, \WObj:=rdkWObj;
	MoveL [[341.480,1210.566,0.000],[0.00000002,0.00000004,1.00000000,-0.00000004],[0,-1,0,0],rdkExtax], rdkSpeed, rdkZone, rdkTool, \WObj:=rdkWObj;
	MoveL [[349.072,1204.231,0.000],[0.00000002,0.00000004,1.00000000,-0.00000004],[0,-1,0,0],rdkExtax], rdkSpeed, rdkZone, rdkTool, \WObj:=rdkWObj;
	MoveL [[356.196,1197.353,0.000],[0.00000002,0.00000004,1.00000000,-0.00000004],[0,-1,0,0],rdkExtax], rdkSpeed, rdkZone, rdkTool, \WObj:=rdkWObj;
	MoveL [[362.827,1189.974,0.000],[0.00000002,0.00000004,1.00000000,-0.00000004],[0,-1,0,0],rdkExtax], rdkSpeed, rdkZone, rdkTool, \WObj:=rdkWObj;
	MoveL [[368.940,1182.135,0.000],[0.00000002,0.00000004,1.00000000,-0.00000004],[0,-1,0,0],rdkExtax], rdkSpeed, rdkZone, rdkTool, \WObj:=rdkWObj;
	MoveL [[374.509,1173.879,0.000],[0.00000002,0.00000004,1.00000000,-0.00000004],[0,-1,0,0],rdkExtax], rdkSpeed, rdkZone, rdkTool, \WObj:=rdkWObj;
	MoveL [[379.509,1165.248,0.000],[0.00000002,0.00000004,1.00000000,-0.00000004],[0,-1,0,0],rdkExtax], rdkSpeed, rdkZone, rdkTool, \WObj:=rdkWObj;
	MoveL [[383.914,1156.283,0.000],[0.00000002,0.00000004,1.00000000,-0.00000004],[0,-1,0,0],rdkExtax], rdkSpeed, rdkZone, rdkTool, \WObj:=rdkWObj;
	MoveL [[387.700,1147.027,0.000],[0.00000002,0.00000004,1.00000000,-0.00000004],[0,-1,0,0],rdkExtax], rdkSpeed, rdkZone, rdkTool, \WObj:=rdkWObj;
	MoveL [[390.840,1137.522,0.000],[0.00000002,0.00000004,1.00000000,-0.00000004],[0,-1,0,0],rdkExtax], rdkSpeed, rdkZone, rdkTool, \WObj:=rdkWObj;
	MoveL [[393.311,1127.810,0.000],[0.00000002,0.00000004,1.00000000,-0.00000004],[0,-1,0,0],rdkExtax], rdkSpeed, rdkZone, rdkTool, \WObj:=rdkWObj;
	MoveL [[395.085,1117.933,0.000],[0.00000002,0.00000004,1.00000000,-0.00000004],[0,-1,0,0],rdkExtax], rdkSpeed, rdkZone, rdkTool, \WObj:=rdkWObj;
	MoveL [[396.139,1107.933,0.000],[0.00000002,0.00000004,1.00000000,-0.00000004],[0,-1,0,0],rdkExtax], rdkSpeed, rdkZone, rdkTool, \WObj:=rdkWObj;
	MoveL [[396.446,1097.851,0.000],[0.00000002,0.00000004,1.00000000,-0.00000004],[0,-1,0,0],rdkExtax], rdkSpeed, rdkZone, rdkTool, \WObj:=rdkWObj;
	MoveL [[395.982,1087.731,0.000],[0.00000002,0.00000004,1.00000000,-0.00000004],[0,-1,0,0],rdkExtax], rdkSpeed, rdkZone, rdkTool, \WObj:=rdkWObj;
	MoveL [[394.721,1077.614,0.000],[0.00000002,0.00000004,1.00000000,-0.00000004],[0,-1,0,0],rdkExtax], rdkSpeed, rdkZone, rdkTool, \WObj:=rdkWObj;
	MoveL [[392.638,1067.542,0.000],[0.00000002,0.00000004,1.00000000,-0.00000004],[0,-1,0,0],rdkExtax], rdkSpeed, rdkZone, rdkTool, \WObj:=rdkWObj;
	MoveL [[389.707,1057.557,0.000],[0.00000002,0.00000004,1.00000000,-0.00000004],[0,-1,0,0],rdkExtax], rdkSpeed, rdkZone, rdkTool, \WObj:=rdkWObj;
	MoveL [[386.802,1047.137,0.000],[0.00000002,0.00000004,1.00000000,-0.00000004],[0,-1,0,0],rdkExtax], rdkSpeed, rdkZone, rdkTool, \WObj:=rdkWObj;
	MoveL [[383.087,1037.304,0.000],[0.00000002,0.00000004,1.00000000,-0.00000004],[0,-1,0,0],rdkExtax], rdkSpeed, rdkZone, rdkTool, \WObj:=rdkWObj;
	MoveL [[378.597,1028.074,0.000],[0.00000002,0.00000004,1.00000000,-0.00000004],[0,-1,0,0],rdkExtax], rdkSpeed, rdkZone, rdkTool, \WObj:=rdkWObj;
	MoveL [[373.381,1019.447,0.000],[0.00000002,0.00000004,1.00000000,-0.00000004],[0,-1,0,0],rdkExtax], rdkSpeed, rdkZone, rdkTool, \WObj:=rdkWObj;
	MoveL [[367.488,1011.425,0.000],[0.00000002,0.00000004,1.00000000,-0.00000004],[0,-1,0,0],rdkExtax], rdkSpeed, rdkZone, rdkTool, \WObj:=rdkWObj;
	MoveL [[360.970,1004.009,0.000],[0.00000002,0.00000004,1.00000000,-0.00000004],[0,-1,0,0],rdkExtax], rdkSpeed, rdkZone, rdkTool, \WObj:=rdkWObj;
	MoveL [[353.875,997.200,0.000],[0.00000002,0.00000004,1.00000000,-0.00000004],[0,-1,0,0],rdkExtax], rdkSpeed, rdkZone, rdkTool, \WObj:=rdkWObj;
	MoveL [[346.254,991.000,0.000],[0.00000002,0.00000004,1.00000000,-0.00000004],[0,-1,0,0],rdkExtax], rdkSpeed, rdkZone, rdkTool, \WObj:=rdkWObj;
	MoveL [[338.156,985.410,0.000],[0.00000002,0.00000004,1.00000000,-0.00000004],[0,-1,0,0],rdkExtax], rdkSpeed, rdkZone, rdkTool, \WObj:=rdkWObj;
	MoveL [[329.631,980.430,0.000],[0.00000002,0.00000004,1.00000000,-0.00000004],[0,-1,0,0],rdkExtax], rdkSpeed, rdkZone, rdkTool, \WObj:=rdkWObj;
	MoveL [[320.730,976.063,0.000],[0.00000002,0.00000004,1.00000000,-0.00000004],[0,-1,0,0],rdkExtax], rdkSpeed, rdkZone, rdkTool, \WObj:=rdkWObj;
	MoveL [[311.501,972.308,0.000],[0.00000002,0.00000004,1.00000000,-0.00000004],[0,-1,0,0],rdkExtax], rdkSpeed, rdkZone, rdkTool, \WObj:=rdkWObj;
	MoveL [[301.994,969.169,0.000],[0.00000002,0.00000004,1.00000000,-0.00000004],[0,-1,0,0],rdkExtax], rdkSpeed, rdkZone, rdkTool, \WObj:=rdkWObj;
	MoveL [[292.261,966.645,0.000],[0.00000002,0.00000004,1.00000000,-0.00000004],[0,-1,0,0],rdkExtax], rdkSpeed, rdkZone, rdkTool, \WObj:=rdkWObj;
	MoveL [[282.349,964.738,0.000],[0.00000002,0.00000004,1.00000000,-0.00000004],[0,-1,0,0],rdkExtax], rdkSpeed, rdkZone, rdkTool, \WObj:=rdkWObj;
	MoveL [[272.310,963.449,0.000],[0.00000002,0.00000004,1.00000000,-0.00000004],[0,-1,0,0],rdkExtax], rdkSpeed, rdkZone, rdkTool, \WObj:=rdkWObj;
	MoveL [[262.193,962.780,0.000],[0.00000002,0.00000004,1.00000000,-0.00000004],[0,-1,0,0],rdkExtax], rdkSpeed, rdkZone, rdkTool, \WObj:=rdkWObj;
	MoveL [[252.047,962.731,0.000],[0.00000002,0.00000004,1.00000000,-0.00000004],[0,-1,0,0],rdkExtax], rdkSpeed, rdkZone, rdkTool, \WObj:=rdkWObj;
	MoveL [[241.924,963.304,0.000],[0.00000002,0.00000004,1.00000000,-0.00000004],[0,-1,0,0],rdkExtax], rdkSpeed, rdkZone, rdkTool, \WObj:=rdkWObj;
	MoveL [[231.871,964.500,0.000],[0.00000002,0.00000004,1.00000000,-0.00000004],[0,-1,0,0],rdkExtax], rdkSpeed, rdkZone, rdkTool, \WObj:=rdkWObj;
	MoveL [[221.941,966.321,0.000],[0.00000002,0.00000004,1.00000000,-0.00000004],[0,-1,0,0],rdkExtax], rdkSpeed, rdkZone, rdkTool, \WObj:=rdkWObj;
	MoveL [[212.181,968.766,0.000],[0.00000002,0.00000004,1.00000000,-0.00000004],[0,-1,0,0],rdkExtax], rdkSpeed, rdkZone, rdkTool, \WObj:=rdkWObj;
	MoveL [[202.642,971.839,0.000],[0.00000002,0.00000004,1.00000000,-0.00000004],[0,-1,0,0],rdkExtax], rdkSpeed, rdkZone, rdkTool, \WObj:=rdkWObj;
	MoveL [[193.374,975.539,0.000],[0.00000002,0.00000004,1.00000000,-0.00000004],[0,-1,0,0],rdkExtax], rdkSpeed, rdkZone, rdkTool, \WObj:=rdkWObj;
	MoveL [[184.427,979.868,0.000],[0.00000002,0.00000004,1.00000000,-0.00000004],[0,-1,0,0],rdkExtax], rdkSpeed, rdkZone, rdkTool, \WObj:=rdkWObj;
	MoveL [[175.851,984.828,0.000],[0.00000002,0.00000004,1.00000000,-0.00000004],[0,-1,0,0],rdkExtax], rdkSpeed, rdkZone, rdkTool, \WObj:=rdkWObj;
	MoveL [[167.695,990.419,0.000],[0.00000002,0.00000004,1.00000000,-0.00000004],[0,-1,0,0],rdkExtax], rdkSpeed, rdkZone, rdkTool, \WObj:=rdkWObj;
	MoveL [[160.009,996.643,0.000],[0.00000002,0.00000004,1.00000000,-0.00000004],[0,-1,0,0],rdkExtax], rdkSpeed, rdkZone, rdkTool, \WObj:=rdkWObj;
	MoveL [[152.843,1003.501,0.000],[0.00000002,0.00000004,1.00000000,-0.00000004],[0,-1,0,0],rdkExtax], rdkSpeed, rdkZone, rdkTool, \WObj:=rdkWObj;
	MoveL [[146.247,1010.993,0.000],[0.00000002,0.00000004,1.00000000,-0.00000004],[0,-1,0,0],rdkExtax], rdkSpeed, rdkZone, rdkTool, \WObj:=rdkWObj;
	MoveL [[140.270,1019.123,0.000],[0.00000002,0.00000004,1.00000000,-0.00000004],[0,-1,0,0],rdkExtax], rdkSpeed, rdkZone, rdkTool, \WObj:=rdkWObj;
	MoveL [[134.964,1027.889,0.000],[0.00000002,0.00000004,1.00000000,-0.00000004],[0,-1,0,0],rdkExtax], rdkSpeed, rdkZone, rdkTool, \WObj:=rdkWObj;
	MoveL [[130.376,1037.295,0.000],[0.00000002,0.00000004,1.00000000,-0.00000004],[0,-1,0,0],rdkExtax], rdkSpeed, rdkZone, rdkTool, \WObj:=rdkWObj;
	MoveL [[126.410,1047.014,0.000],[0.00000002,0.00000004,1.00000000,-0.00000004],[0,-1,0,0],rdkExtax], rdkSpeed, rdkZone, rdkTool, \WObj:=rdkWObj;
	MoveL [[123.053,1056.667,0.000],[0.00000002,0.00000004,1.00000000,-0.00000004],[0,-1,0,0],rdkExtax], rdkSpeed, rdkZone, rdkTool, \WObj:=rdkWObj;
	MoveL [[120.473,1066.499,0.000],[0.00000002,0.00000004,1.00000000,-0.00000004],[0,-1,0,0],rdkExtax], rdkSpeed, rdkZone, rdkTool, \WObj:=rdkWObj;
	MoveL [[118.654,1076.466,0.000],[0.00000002,0.00000004,1.00000000,-0.00000004],[0,-1,0,0],rdkExtax], rdkSpeed, rdkZone, rdkTool, \WObj:=rdkWObj;
	MoveL [[117.577,1086.520,0.000],[0.00000002,0.00000004,1.00000000,-0.00000004],[0,-1,0,0],rdkExtax], rdkSpeed, rdkZone, rdkTool, \WObj:=rdkWObj;
	MoveL [[117.225,1096.615,0.000],[0.00000002,0.00000004,1.00000000,-0.00000004],[0,-1,0,0],rdkExtax], rdkSpeed, rdkZone, rdkTool, \WObj:=rdkWObj;
	MoveL [[117.581,1106.704,0.000],[0.00000002,0.00000004,1.00000000,-0.00000004],[0,-1,0,0],rdkExtax], rdkSpeed, rdkZone, rdkTool, \WObj:=rdkWObj;
	MoveL [[118.627,1116.741,0.000],[0.00000002,0.00000004,1.00000000,-0.00000004],[0,-1,0,0],rdkExtax], rdkSpeed, rdkZone, rdkTool, \WObj:=rdkWObj;
	MoveL [[120.346,1126.679,0.000],[0.00000002,0.00000004,1.00000000,-0.00000004],[0,-1,0,0],rdkExtax], rdkSpeed, rdkZone, rdkTool, \WObj:=rdkWObj;
	MoveL [[122.721,1136.471,0.000],[0.00000002,0.00000004,1.00000000,-0.00000004],[0,-1,0,0],rdkExtax], rdkSpeed, rdkZone, rdkTool, \WObj:=rdkWObj;
	MoveL [[125.734,1146.071,0.000],[0.00000002,0.00000004,1.00000000,-0.00000004],[0,-1,0,0],rdkExtax], rdkSpeed, rdkZone, rdkTool, \WObj:=rdkWObj;
	MoveL [[129.368,1155.433,0.000],[0.00000002,0.00000004,1.00000000,-0.00000004],[0,-1,0,0],rdkExtax], rdkSpeed, rdkZone, rdkTool, \WObj:=rdkWObj;
	MoveL [[133.606,1164.509,0.000],[0.00000002,0.00000004,1.00000000,-0.00000004],[0,-1,0,0],rdkExtax], rdkSpeed, rdkZone, rdkTool, \WObj:=rdkWObj;
	MoveL [[138.430,1173.254,0.000],[0.00000002,0.00000004,1.00000000,-0.00000004],[0,-1,0,0],rdkExtax], rdkSpeed, rdkZone, rdkTool, \WObj:=rdkWObj;
	MoveL [[143.822,1181.621,0.000],[0.00000002,0.00000004,1.00000000,-0.00000004],[0,-1,0,0],rdkExtax], rdkSpeed, rdkZone, rdkTool, \WObj:=rdkWObj;
	MoveL [[149.767,1189.563,0.000],[0.00000002,0.00000004,1.00000000,-0.00000004],[0,-1,0,0],rdkExtax], rdkSpeed, rdkZone, rdkTool, \WObj:=rdkWObj;
	MoveL [[156.245,1197.033,0.000],[0.00000002,0.00000004,1.00000000,-0.00000004],[0,-1,0,0],rdkExtax], rdkSpeed, rdkZone, rdkTool, \WObj:=rdkWObj;
	MoveL [[163.240,1203.986,0.000],[0.00000002,0.00000004,1.00000000,-0.00000004],[0,-1,0,0],rdkExtax], rdkSpeed, rdkZone, rdkTool, \WObj:=rdkWObj;
	MoveL [[170.734,1210.374,0.000],[0.00000002,0.00000004,1.00000000,-0.00000004],[0,-1,0,0],rdkExtax], rdkSpeed, rdkZone, rdkTool, \WObj:=rdkWObj;
	MoveL [[178.710,1216.151,0.000],[0.00000002,0.00000004,1.00000000,-0.00000004],[0,-1,0,0],rdkExtax], rdkSpeed, rdkZone, rdkTool, \WObj:=rdkWObj;
	MoveL [[187.151,1221.270,0.000],[0.00000002,0.00000004,1.00000000,-0.00000004],[0,-1,0,0],rdkExtax], rdkSpeed, rdkZone, rdkTool, \WObj:=rdkWObj;
	MoveL [[196.040,1225.686,0.000],[0.00000002,0.00000004,1.00000000,-0.00000004],[0,-1,0,0],rdkExtax], rdkSpeed, rdkZone, rdkTool, \WObj:=rdkWObj;
	MoveL [[205.358,1229.350,0.000],[0.00000002,0.00000004,1.00000000,-0.00000004],[0,-1,0,0],rdkExtax], rdkSpeed, rdkZone, rdkTool, \WObj:=rdkWObj;
	MoveL [[215.088,1232.218,0.000],[0.00000002,0.00000004,1.00000000,-0.00000004],[0,-1,0,0],rdkExtax], rdkSpeed, rdkZone, rdkTool, \WObj:=rdkWObj;
	MoveL [[225.214,1234.241,0.000],[0.00000002,0.00000004,1.00000000,-0.00000004],[0,-1,0,0],rdkExtax], rdkSpeed, rdkZone, rdkTool, \WObj:=rdkWObj;
	MoveL [[235.717,1235.374,0.000],[0.00000002,0.00000004,1.00000000,-0.00000004],[0,-1,0,0],rdkExtax], rdkSpeed, rdkZone, rdkTool, \WObj:=rdkWObj;
	MoveL [[246.155,1235.788,0.000],[0.00000002,0.00000004,1.00000000,-0.00000004],[0,-1,0,0],rdkExtax], rdkSpeed, rdkZone, rdkTool, \WObj:=rdkWObj;
	MoveL [[256.222,1236.186,0.000],[0.00000002,0.00000004,1.00000000,-0.00000004],[0,-1,0,0],rdkExtax], rdkSpeed, rdkZone, rdkTool, \WObj:=rdkWObj;
	MoveL [[242.819,1146.566,0.000],[0.00000002,0.00000004,1.00000000,-0.00000004],[0,-1,0,0],rdkExtax], rdkSpeed, rdkZone, rdkTool, \WObj:=rdkWObj;
	MoveL [[231.534,1143.744,0.000],[0.00000002,0.00000004,1.00000000,-0.00000004],[0,-1,0,0],rdkExtax], rdkSpeed, rdkZone, rdkTool, \WObj:=rdkWObj;
	MoveL [[222.396,1139.151,0.000],[0.00000002,0.00000004,1.00000000,-0.00000004],[0,-1,0,0],rdkExtax], rdkSpeed, rdkZone, rdkTool, \WObj:=rdkWObj;
	MoveL [[215.306,1133.074,0.000],[0.00000002,0.00000004,1.00000000,-0.00000004],[0,-1,0,0],rdkExtax], rdkSpeed, rdkZone, rdkTool, \WObj:=rdkWObj;
	MoveL [[210.163,1125.799,0.000],[0.00000002,0.00000004,1.00000000,-0.00000004],[0,-1,0,0],rdkExtax], rdkSpeed, rdkZone, rdkTool, \WObj:=rdkWObj;
	MoveL [[206.867,1117.615,0.000],[0.00000002,0.00000004,1.00000000,-0.00000004],[0,-1,0,0],rdkExtax], rdkSpeed, rdkZone, rdkTool, \WObj:=rdkWObj;
	MoveL [[205.316,1108.809,0.000],[0.00000002,0.00000004,1.00000000,-0.00000004],[0,-1,0,0],rdkExtax], rdkSpeed, rdkZone, rdkTool, \WObj:=rdkWObj;
	MoveL [[205.410,1099.667,0.000],[0.00000002,0.00000004,1.00000000,-0.00000004],[0,-1,0,0],rdkExtax], rdkSpeed, rdkZone, rdkTool, \WObj:=rdkWObj;
	MoveL [[207.048,1090.476,0.000],[0.00000002,0.00000004,1.00000000,-0.00000004],[0,-1,0,0],rdkExtax], rdkSpeed, rdkZone, rdkTool, \WObj:=rdkWObj;
	MoveL [[210.130,1081.524,0.000],[0.00000002,0.00000004,1.00000000,-0.00000004],[0,-1,0,0],rdkExtax], rdkSpeed, rdkZone, rdkTool, \WObj:=rdkWObj;
	MoveL [[214.555,1073.099,0.000],[0.00000002,0.00000004,1.00000000,-0.00000004],[0,-1,0,0],rdkExtax], rdkSpeed, rdkZone, rdkTool, \WObj:=rdkWObj;
	MoveL [[220.222,1065.486,0.000],[0.00000002,0.00000004,1.00000000,-0.00000004],[0,-1,0,0],rdkExtax], rdkSpeed, rdkZone, rdkTool, \WObj:=rdkWObj;
	MoveL [[227.031,1058.974,0.000],[0.00000002,0.00000004,1.00000000,-0.00000004],[0,-1,0,0],rdkExtax], rdkSpeed, rdkZone, rdkTool, \WObj:=rdkWObj;
	MoveL [[234.881,1053.849,0.000],[0.00000002,0.00000004,1.00000000,-0.00000004],[0,-1,0,0],rdkExtax], rdkSpeed, rdkZone, rdkTool, \WObj:=rdkWObj;
	MoveL [[243.671,1050.399,0.000],[0.00000002,0.00000004,1.00000000,-0.00000004],[0,-1,0,0],rdkExtax], rdkSpeed, rdkZone, rdkTool, \WObj:=rdkWObj;
	MoveL [[253.301,1048.911,0.000],[0.00000002,0.00000004,1.00000000,-0.00000004],[0,-1,0,0],rdkExtax], rdkSpeed, rdkZone, rdkTool, \WObj:=rdkWObj;
	MoveL [[263.670,1049.671,0.000],[0.00000002,0.00000004,1.00000000,-0.00000004],[0,-1,0,0],rdkExtax], rdkSpeed, rdkZone, rdkTool, \WObj:=rdkWObj;
	MoveL [[274.677,1052.968,0.000],[0.00000002,0.00000004,1.00000000,-0.00000004],[0,-1,0,0],rdkExtax], rdkSpeed, rdkZone, rdkTool, \WObj:=rdkWObj;
	MoveL [[286.183,1058.997,0.000],[0.00000002,0.00000004,1.00000000,-0.00000004],[0,-1,0,0],rdkExtax], rdkSpeed, rdkZone, rdkTool, \WObj:=rdkWObj;
	MoveL [[295.750,1065.335,0.000],[0.00000002,0.00000004,1.00000000,-0.00000004],[0,-1,0,0],rdkExtax], rdkSpeed, rdkZone, rdkTool, \WObj:=rdkWObj;
	MoveL [[302.816,1072.939,0.000],[0.00000002,0.00000004,1.00000000,-0.00000004],[0,-1,0,0],rdkExtax], rdkSpeed, rdkZone, rdkTool, \WObj:=rdkWObj;
	MoveL [[307.525,1081.484,0.000],[0.00000002,0.00000004,1.00000000,-0.00000004],[0,-1,0,0],rdkExtax], rdkSpeed, rdkZone, rdkTool, \WObj:=rdkWObj;
	MoveL [[310.018,1090.646,0.000],[0.00000002,0.00000004,1.00000000,-0.00000004],[0,-1,0,0],rdkExtax], rdkSpeed, rdkZone, rdkTool, \WObj:=rdkWObj;
	MoveL [[310.438,1100.100,0.000],[0.00000002,0.00000004,1.00000000,-0.00000004],[0,-1,0,0],rdkExtax], rdkSpeed, rdkZone, rdkTool, \WObj:=rdkWObj;
	MoveL [[308.928,1109.522,0.000],[0.00000002,0.00000004,1.00000000,-0.00000004],[0,-1,0,0],rdkExtax], rdkSpeed, rdkZone, rdkTool, \WObj:=rdkWObj;
	MoveL [[305.630,1118.588,0.000],[0.00000002,0.00000004,1.00000000,-0.00000004],[0,-1,0,0],rdkExtax], rdkSpeed, rdkZone, rdkTool, \WObj:=rdkWObj;
	MoveL [[300.686,1126.972,0.000],[0.00000002,0.00000004,1.00000000,-0.00000004],[0,-1,0,0],rdkExtax], rdkSpeed, rdkZone, rdkTool, \WObj:=rdkWObj;
	MoveL [[294.240,1134.352,0.000],[0.00000002,0.00000004,1.00000000,-0.00000004],[0,-1,0,0],rdkExtax], rdkSpeed, rdkZone, rdkTool, \WObj:=rdkWObj;
	MoveL [[286.433,1140.402,0.000],[0.00000002,0.00000004,1.00000000,-0.00000004],[0,-1,0,0],rdkExtax], rdkSpeed, rdkZone, rdkTool, \WObj:=rdkWObj;
	MoveL [[277.409,1144.798,0.000],[0.00000002,0.00000004,1.00000000,-0.00000004],[0,-1,0,0],rdkExtax], rdkSpeed, rdkZone, rdkTool, \WObj:=rdkWObj;
	MoveL [[267.309,1147.216,0.000],[0.00000002,0.00000004,1.00000000,-0.00000004],[0,-1,0,0],rdkExtax], rdkSpeed, rdkZone, rdkTool, \WObj:=rdkWObj;
	MoveL [[256.276,1147.331,0.000],[0.00000002,0.00000004,1.00000000,-0.00000004],[0,-1,0,0],rdkExtax], rdkSpeed, rdkZone, rdkTool, \WObj:=rdkWObj;
	MoveL [[256.276,1147.331,100.000],[0.00000002,0.00000004,1.00000000,-0.00000004],[0,-1,0,0],rdkExtax], rdkSpeed, rdkZone, rdkTool, \WObj:=rdkWObj;
	MoveL [[197.489,1624.671,100.000],[0.00000002,0.00000004,1.00000000,-0.00000004],[0,-1,0,0],rdkExtax], rdkSpeed, rdkZone, rdkTool, \WObj:=rdkWObj;
	TPWrite "Drawing path2998";
	SetColorRGB(0.000,0.294,0.431);
	MoveL [[197.489,1624.671,0.000],[0.00000002,0.00000004,1.00000000,-0.00000004],[0,-1,0,0],rdkExtax], rdkSpeed, rdkZone, rdkTool, \WObj:=rdkWObj;
	MoveL [[207.584,1624.802,0.000],[0.00000002,0.00000004,1.00000000,-0.00000004],[0,-1,0,0],rdkExtax], rdkSpeed, rdkZone, rdkTool, \WObj:=rdkWObj;
	MoveL [[217.661,1624.358,0.000],[0.00000002,0.00000004,1.00000000,-0.00000004],[0,-1,0,0],rdkExtax], rdkSpeed, rdkZone, rdkTool, \WObj:=rdkWObj;
	MoveL [[227.695,1623.353,0.000],[0.00000002,0.00000004,1.00000000,-0.00000004],[0,-1,0,0],rdkExtax], rdkSpeed, rdkZone, rdkTool, \WObj:=rdkWObj;
	MoveL [[237.659,1621.803,0.000],[0.00000002,0.00000004,1.00000000,-0.00000004],[0,-1,0,0],rdkExtax], rdkSpeed, rdkZone, rdkTool, \WObj:=rdkWObj;
	MoveL [[247.529,1619.721,0.000],[0.00000002,0.00000004,1.00000000,-0.00000004],[0,-1,0,0],rdkExtax], rdkSpeed, rdkZone, rdkTool, \WObj:=rdkWObj;
	MoveL [[257.281,1617.123,0.000],[0.00000002,0.00000004,1.00000000,-0.00000004],[0,-1,0,0],rdkExtax], rdkSpeed, rdkZone, rdkTool, \WObj:=rdkWObj;
	MoveL [[266.887,1614.022,0.000],[0.00000002,0.00000004,1.00000000,-0.00000004],[0,-1,0,0],rdkExtax], rdkSpeed, rdkZone, rdkTool, \WObj:=rdkWObj;
	MoveL [[276.324,1610.434,0.000],[0.00000002,0.00000004,1.00000000,-0.00000004],[0,-1,0,0],rdkExtax], rdkSpeed, rdkZone, rdkTool, \WObj:=rdkWObj;
	MoveL [[285.566,1606.374,0.000],[0.00000002,0.00000004,1.00000000,-0.00000004],[0,-1,0,0],rdkExtax], rdkSpeed, rdkZone, rdkTool, \WObj:=rdkWObj;
	MoveL [[294.589,1601.855,0.000],[0.00000002,0.00000004,1.00000000,-0.00000004],[0,-1,0,0],rdkExtax], rdkSpeed, rdkZone, rdkTool, \WObj:=rdkWObj;
	MoveL [[303.366,1596.892,0.000],[0.00000002,0.00000004,1.00000000,-0.00000004],[0,-1,0,0],rdkExtax], rdkSpeed, rdkZone, rdkTool, \WObj:=rdkWObj;
	MoveL [[311.872,1591.500,0.000],[0.00000002,0.00000004,1.00000000,-0.00000004],[0,-1,0,0],rdkExtax], rdkSpeed, rdkZone, rdkTool, \WObj:=rdkWObj;
	MoveL [[320.083,1585.694,0.000],[0.00000002,0.00000004,1.00000000,-0.00000004],[0,-1,0,0],rdkExtax], rdkSpeed, rdkZone, rdkTool, \WObj:=rdkWObj;
	MoveL [[327.974,1579.487,0.000],[0.00000002,0.00000004,1.00000000,-0.00000004],[0,-1,0,0],rdkExtax], rdkSpeed, rdkZone, rdkTool, \WObj:=rdkWObj;
	MoveL [[335.518,1572.896,0.000],[0.00000002,0.00000004,1.00000000,-0.00000004],[0,-1,0,0],rdkExtax], rdkSpeed, rdkZone, rdkTool, \WObj:=rdkWObj;
	MoveL [[342.691,1565.934,0.000],[0.00000002,0.00000004,1.00000000,-0.00000004],[0,-1,0,0],rdkExtax], rdkSpeed, rdkZone, rdkTool, \WObj:=rdkWObj;
	MoveL [[349.468,1558.615,0.000],[0.00000002,0.00000004,1.00000000,-0.00000004],[0,-1,0,0],rdkExtax], rdkSpeed, rdkZone, rdkTool, \WObj:=rdkWObj;
	MoveL [[355.824,1550.955,0.000],[0.00000002,0.00000004,1.00000000,-0.00000004],[0,-1,0,0],rdkExtax], rdkSpeed, rdkZone, rdkTool, \WObj:=rdkWObj;
	MoveL [[361.733,1542.969,0.000],[0.00000002,0.00000004,1.00000000,-0.00000004],[0,-1,0,0],rdkExtax], rdkSpeed, rdkZone, rdkTool, \WObj:=rdkWObj;
	MoveL [[367.170,1534.670,0.000],[0.00000002,0.00000004,1.00000000,-0.00000004],[0,-1,0,0],rdkExtax], rdkSpeed, rdkZone, rdkTool, \WObj:=rdkWObj;
	MoveL [[372.109,1526.073,0.000],[0.00000002,0.00000004,1.00000000,-0.00000004],[0,-1,0,0],rdkExtax], rdkSpeed, rdkZone, rdkTool, \WObj:=rdkWObj;
	MoveL [[376.527,1517.193,0.000],[0.00000002,0.00000004,1.00000000,-0.00000004],[0,-1,0,0],rdkExtax], rdkSpeed, rdkZone, rdkTool, \WObj:=rdkWObj;
	MoveL [[380.397,1508.045,0.000],[0.00000002,0.00000004,1.00000000,-0.00000004],[0,-1,0,0],rdkExtax], rdkSpeed, rdkZone, rdkTool, \WObj:=rdkWObj;
	MoveL [[383.695,1498.643,0.000],[0.00000002,0.00000004,1.00000000,-0.00000004],[0,-1,0,0],rdkExtax], rdkSpeed, rdkZone, rdkTool, \WObj:=rdkWObj;
	MoveL [[386.395,1489.001,0.000],[0.00000002,0.00000004,1.00000000,-0.00000004],[0,-1,0,0],rdkExtax], rdkSpeed, rdkZone, rdkTool, \WObj:=rdkWObj;
	MoveL [[388.472,1479.135,0.000],[0.00000002,0.00000004,1.00000000,-0.00000004],[0,-1,0,0],rdkExtax], rdkSpeed, rdkZone, rdkTool, \WObj:=rdkWObj;
	MoveL [[389.900,1469.059,0.000],[0.00000002,0.00000004,1.00000000,-0.00000004],[0,-1,0,0],rdkExtax], rdkSpeed, rdkZone, rdkTool, \WObj:=rdkWObj;
	MoveL [[390.656,1458.787,0.000],[0.00000002,0.00000004,1.00000000,-0.00000004],[0,-1,0,0],rdkExtax], rdkSpeed, rdkZone, rdkTool, \WObj:=rdkWObj;
	MoveL [[390.713,1448.334,0.000],[0.00000002,0.00000004,1.00000000,-0.00000004],[0,-1,0,0],rdkExtax], rdkSpeed, rdkZone, rdkTool, \WObj:=rdkWObj;
	MoveL [[389.641,1438.896,0.000],[0.00000002,0.00000004,1.00000000,-0.00000004],[0,-1,0,0],rdkExtax], rdkSpeed, rdkZone, rdkTool, \WObj:=rdkWObj;
	MoveL [[388.973,1429.183,0.000],[0.00000002,0.00000004,1.00000000,-0.00000004],[0,-1,0,0],rdkExtax], rdkSpeed, rdkZone, rdkTool, \WObj:=rdkWObj;
	MoveL [[388.821,1418.981,0.000],[0.00000002,0.00000004,1.00000000,-0.00000004],[0,-1,0,0],rdkExtax], rdkSpeed, rdkZone, rdkTool, \WObj:=rdkWObj;
	MoveL [[389.077,1408.387,0.000],[0.00000002,0.00000004,1.00000000,-0.00000004],[0,-1,0,0],rdkExtax], rdkSpeed, rdkZone, rdkTool, \WObj:=rdkWObj;
	MoveL [[389.634,1397.495,0.000],[0.00000002,0.00000004,1.00000000,-0.00000004],[0,-1,0,0],rdkExtax], rdkSpeed, rdkZone, rdkTool, \WObj:=rdkWObj;
	MoveL [[390.382,1386.400,0.000],[0.00000002,0.00000004,1.00000000,-0.00000004],[0,-1,0,0],rdkExtax], rdkSpeed, rdkZone, rdkTool, \WObj:=rdkWObj;
	MoveL [[391.214,1375.196,0.000],[0.00000002,0.00000004,1.00000000,-0.00000004],[0,-1,0,0],rdkExtax], rdkSpeed, rdkZone, rdkTool, \WObj:=rdkWObj;
	MoveL [[392.022,1363.978,0.000],[0.00000002,0.00000004,1.00000000,-0.00000004],[0,-1,0,0],rdkExtax], rdkSpeed, rdkZone, rdkTool, \WObj:=rdkWObj;
	MoveL [[392.698,1352.840,0.000],[0.00000002,0.00000004,1.00000000,-0.00000004],[0,-1,0,0],rdkExtax], rdkSpeed, rdkZone, rdkTool, \WObj:=rdkWObj;
	MoveL [[393.134,1341.879,0.000],[0.00000002,0.00000004,1.00000000,-0.00000004],[0,-1,0,0],rdkExtax], rdkSpeed, rdkZone, rdkTool, \WObj:=rdkWObj;
	MoveL [[393.221,1331.187,0.000],[0.00000002,0.00000004,1.00000000,-0.00000004],[0,-1,0,0],rdkExtax], rdkSpeed, rdkZone, rdkTool, \WObj:=rdkWObj;
	MoveL [[392.852,1320.860,0.000],[0.00000002,0.00000004,1.00000000,-0.00000004],[0,-1,0,0],rdkExtax], rdkSpeed, rdkZone, rdkTool, \WObj:=rdkWObj;
	MoveL [[391.919,1310.993,0.000],[0.00000002,0.00000004,1.00000000,-0.00000004],[0,-1,0,0],rdkExtax], rdkSpeed, rdkZone, rdkTool, \WObj:=rdkWObj;
	MoveL [[390.314,1301.680,0.000],[0.00000002,0.00000004,1.00000000,-0.00000004],[0,-1,0,0],rdkExtax], rdkSpeed, rdkZone, rdkTool, \WObj:=rdkWObj;
	MoveL [[387.928,1293.016,0.000],[0.00000002,0.00000004,1.00000000,-0.00000004],[0,-1,0,0],rdkExtax], rdkSpeed, rdkZone, rdkTool, \WObj:=rdkWObj;
	MoveL [[384.654,1285.096,0.000],[0.00000002,0.00000004,1.00000000,-0.00000004],[0,-1,0,0],rdkExtax], rdkSpeed, rdkZone, rdkTool, \WObj:=rdkWObj;
	MoveL [[380.383,1278.014,0.000],[0.00000002,0.00000004,1.00000000,-0.00000004],[0,-1,0,0],rdkExtax], rdkSpeed, rdkZone, rdkTool, \WObj:=rdkWObj;
	MoveL [[374.724,1272.289,0.000],[0.00000002,0.00000004,1.00000000,-0.00000004],[0,-1,0,0],rdkExtax], rdkSpeed, rdkZone, rdkTool, \WObj:=rdkWObj;
	MoveL [[364.664,1272.765,0.000],[0.00000002,0.00000004,1.00000000,-0.00000004],[0,-1,0,0],rdkExtax], rdkSpeed, rdkZone, rdkTool, \WObj:=rdkWObj;
	MoveL [[354.605,1273.206,0.000],[0.00000002,0.00000004,1.00000000,-0.00000004],[0,-1,0,0],rdkExtax], rdkSpeed, rdkZone, rdkTool, \WObj:=rdkWObj;
	MoveL [[344.545,1273.613,0.000],[0.00000002,0.00000004,1.00000000,-0.00000004],[0,-1,0,0],rdkExtax], rdkSpeed, rdkZone, rdkTool, \WObj:=rdkWObj;
	MoveL [[334.485,1273.987,0.000],[0.00000002,0.00000004,1.00000000,-0.00000004],[0,-1,0,0],rdkExtax], rdkSpeed, rdkZone, rdkTool, \WObj:=rdkWObj;
	MoveL [[324.425,1274.329,0.000],[0.00000002,0.00000004,1.00000000,-0.00000004],[0,-1,0,0],rdkExtax], rdkSpeed, rdkZone, rdkTool, \WObj:=rdkWObj;
	MoveL [[314.366,1274.638,0.000],[0.00000002,0.00000004,1.00000000,-0.00000004],[0,-1,0,0],rdkExtax], rdkSpeed, rdkZone, rdkTool, \WObj:=rdkWObj;
	MoveL [[304.306,1274.917,0.000],[0.00000002,0.00000004,1.00000000,-0.00000004],[0,-1,0,0],rdkExtax], rdkSpeed, rdkZone, rdkTool, \WObj:=rdkWObj;
	MoveL [[294.246,1275.164,0.000],[0.00000002,0.00000004,1.00000000,-0.00000004],[0,-1,0,0],rdkExtax], rdkSpeed, rdkZone, rdkTool, \WObj:=rdkWObj;
	MoveL [[284.186,1275.382,0.000],[0.00000002,0.00000004,1.00000000,-0.00000004],[0,-1,0,0],rdkExtax], rdkSpeed, rdkZone, rdkTool, \WObj:=rdkWObj;
	MoveL [[274.126,1275.570,0.000],[0.00000002,0.00000004,1.00000000,-0.00000004],[0,-1,0,0],rdkExtax], rdkSpeed, rdkZone, rdkTool, \WObj:=rdkWObj;
	MoveL [[264.066,1275.729,0.000],[0.00000002,0.00000004,1.00000000,-0.00000004],[0,-1,0,0],rdkExtax], rdkSpeed, rdkZone, rdkTool, \WObj:=rdkWObj;
	MoveL [[254.006,1275.860,0.000],[0.00000002,0.00000004,1.00000000,-0.00000004],[0,-1,0,0],rdkExtax], rdkSpeed, rdkZone, rdkTool, \WObj:=rdkWObj;
	MoveL [[243.946,1275.963,0.000],[0.00000002,0.00000004,1.00000000,-0.00000004],[0,-1,0,0],rdkExtax], rdkSpeed, rdkZone, rdkTool, \WObj:=rdkWObj;
	MoveL [[233.886,1276.038,0.000],[0.00000002,0.00000004,1.00000000,-0.00000004],[0,-1,0,0],rdkExtax], rdkSpeed, rdkZone, rdkTool, \WObj:=rdkWObj;
	MoveL [[223.826,1276.087,0.000],[0.00000002,0.00000004,1.00000000,-0.00000004],[0,-1,0,0],rdkExtax], rdkSpeed, rdkZone, rdkTool, \WObj:=rdkWObj;
	MoveL [[213.766,1276.111,0.000],[0.00000002,0.00000004,1.00000000,-0.00000004],[0,-1,0,0],rdkExtax], rdkSpeed, rdkZone, rdkTool, \WObj:=rdkWObj;
	MoveL [[203.706,1276.108,0.000],[0.00000002,0.00000004,1.00000000,-0.00000004],[0,-1,0,0],rdkExtax], rdkSpeed, rdkZone, rdkTool, \WObj:=rdkWObj;
	MoveL [[193.646,1276.081,0.000],[0.00000002,0.00000004,1.00000000,-0.00000004],[0,-1,0,0],rdkExtax], rdkSpeed, rdkZone, rdkTool, \WObj:=rdkWObj;
	MoveL [[183.586,1276.030,0.000],[0.00000002,0.00000004,1.00000000,-0.00000004],[0,-1,0,0],rdkExtax], rdkSpeed, rdkZone, rdkTool, \WObj:=rdkWObj;
	MoveL [[173.525,1275.955,0.000],[0.00000002,0.00000004,1.00000000,-0.00000004],[0,-1,0,0],rdkExtax], rdkSpeed, rdkZone, rdkTool, \WObj:=rdkWObj;
	MoveL [[163.465,1275.856,0.000],[0.00000002,0.00000004,1.00000000,-0.00000004],[0,-1,0,0],rdkExtax], rdkSpeed, rdkZone, rdkTool, \WObj:=rdkWObj;
	MoveL [[153.405,1275.736,0.000],[0.00000002,0.00000004,1.00000000,-0.00000004],[0,-1,0,0],rdkExtax], rdkSpeed, rdkZone, rdkTool, \WObj:=rdkWObj;
